Yaskawa INFORM job: A_ROOF_SIDE_0617_2_PAINT_36.JBI

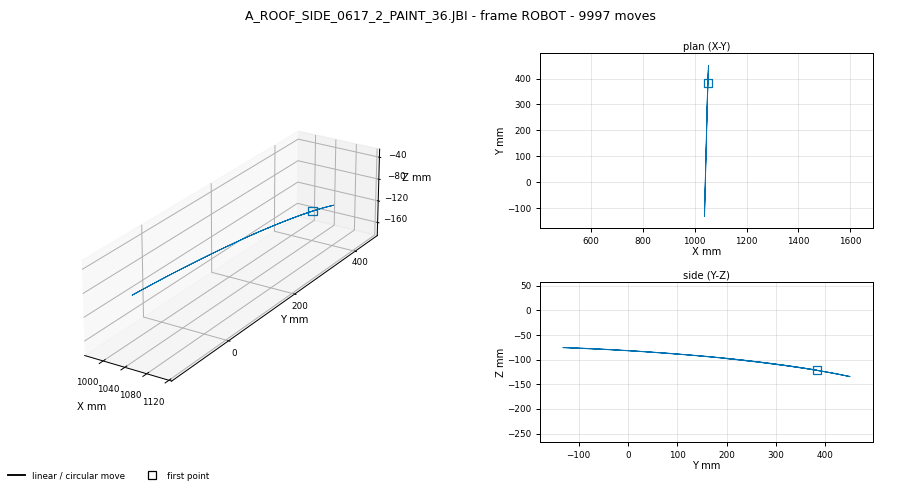
[picture p0: tool path of A_ROOF_SIDE_0617_2_PAINT_36.JBI in frame ROBOT, 9997 of 9997 moves have a stored position in this frame; points joined in program order, loops and branches not executed]
/JOB
//NAME A_ROOF_SIDE_0617_2_PAINT36
//POS
///NPOS 9997,0,0,0,0,0
///TOOL 1
///USER 0
///POSTYPE ROBOT
///RECTAN
///RCONF 1,0,0,0,0,0,0,0,0,0,0,0,0,0,0,0,0,0,0,0,0,0,0,0
C00000=1051.192,382.827,-120.850,173.969,40.523,157.828
C00001=1051.183,382.580,-120.809,173.963,40.517,157.826
C00002=1051.175,382.334,-120.768,173.957,40.511,157.824
C00003=1051.168,382.087,-120.727,173.951,40.505,157.822
C00004=1051.160,381.841,-120.686,173.945,40.499,157.821
C00005=1051.152,381.595,-120.645,173.938,40.493,157.819
C00006=1051.145,381.348,-120.604,173.932,40.487,157.817
C00007=1051.136,381.101,-120.563,173.926,40.481,157.815
C00008=1051.128,380.855,-120.523,173.919,40.475,157.814
C00009=1051.120,380.609,-120.482,173.913,40.469,157.812
C00010=1051.113,380.362,-120.441,173.908,40.463,157.810
C00011=1051.105,380.116,-120.400,173.901,40.458,157.809
C00012=1051.097,379.870,-120.359,173.895,40.452,157.807
C00013=1051.089,379.623,-120.319,173.889,40.446,157.805
C00014=1051.081,379.376,-120.279,173.882,40.440,157.804
C00015=1051.073,379.130,-120.238,173.877,40.434,157.802
C00016=1051.065,378.884,-120.198,173.871,40.429,157.800
C00017=1051.057,378.637,-120.158,173.864,40.423,157.798
C00018=1051.048,378.390,-120.117,173.858,40.417,157.797
C00019=1051.040,378.144,-120.076,173.853,40.412,157.795
C00020=1051.033,377.897,-120.036,173.847,40.406,157.794
C00021=1051.025,377.650,-119.995,173.840,40.400,157.792
C00022=1051.017,377.403,-119.956,173.834,40.395,157.790
C00023=1051.009,377.157,-119.915,173.829,40.389,157.789
C00024=1051.001,376.910,-119.875,173.823,40.383,157.787
C00025=1050.993,376.664,-119.834,173.817,40.378,157.785
C00026=1050.986,376.418,-119.795,173.810,40.372,157.784
C00027=1050.978,376.172,-119.754,173.805,40.367,157.782
C00028=1050.970,375.925,-119.714,173.799,40.361,157.780
C00029=1050.963,375.678,-119.674,173.793,40.356,157.779
C00030=1050.953,375.363,-119.623,173.785,40.348,157.777
C00031=1050.943,375.047,-119.571,173.778,40.341,157.775
C00032=1050.932,374.732,-119.520,173.771,40.334,157.773
C00033=1050.923,374.417,-119.469,173.763,40.327,157.771
C00034=1050.915,374.170,-119.429,173.757,40.321,157.769
C00035=1050.907,373.923,-119.389,173.751,40.316,157.768
C00036=1050.900,373.677,-119.349,173.746,40.310,157.766
C00037=1050.892,373.430,-119.309,173.740,40.305,157.764
C00038=1050.885,373.183,-119.269,173.734,40.300,157.763
C00039=1050.877,372.936,-119.229,173.729,40.294,157.761
C00040=1050.869,372.691,-119.190,173.723,40.288,157.760
C00041=1050.861,372.444,-119.150,173.717,40.283,157.758
C00042=1050.853,372.197,-119.110,173.711,40.278,157.757
C00043=1050.846,371.950,-119.070,173.705,40.272,157.755
C00044=1050.838,371.704,-119.031,173.699,40.267,157.753
C00045=1050.831,371.457,-118.991,173.694,40.262,157.752
C00046=1050.823,371.209,-118.951,173.688,40.256,157.750
C00047=1050.815,370.963,-118.912,173.683,40.251,157.749
C00048=1050.808,370.716,-118.873,173.677,40.246,157.747
C00049=1050.799,370.470,-118.833,173.672,40.240,157.746
C00050=1050.792,370.223,-118.793,173.666,40.235,157.744
C00051=1050.785,369.976,-118.754,173.660,40.230,157.743
C00052=1050.776,369.729,-118.715,173.655,40.225,157.741
C00053=1050.769,369.483,-118.675,173.649,40.219,157.740
C00054=1050.761,369.236,-118.637,173.644,40.214,157.738
C00055=1050.753,368.989,-118.597,173.638,40.209,157.737
C00056=1050.747,368.742,-118.558,173.633,40.204,157.735
C00057=1050.738,368.496,-118.519,173.627,40.199,157.734
C00058=1050.730,368.249,-118.479,173.621,40.193,157.732
C00059=1050.723,368.002,-118.441,173.616,40.188,157.731
C00060=1050.715,367.755,-118.401,173.610,40.183,157.729
C00061=1050.708,367.509,-118.362,173.605,40.178,157.728
C00062=1050.700,367.262,-118.323,173.599,40.173,157.727
C00063=1050.693,367.015,-118.284,173.594,40.167,157.725
C00064=1050.685,366.768,-118.245,173.588,40.163,157.724
C00065=1050.678,366.522,-118.206,173.583,40.157,157.722
C00066=1050.670,366.275,-118.167,173.577,40.152,157.721
C00067=1050.663,366.028,-118.128,173.572,40.147,157.719
C00068=1050.655,365.781,-118.088,173.566,40.142,157.718
C00069=1050.647,365.534,-118.050,173.561,40.137,157.716
C00070=1050.640,365.287,-118.011,173.555,40.132,157.715
C00071=1050.632,365.041,-117.972,173.551,40.127,157.714
C00072=1050.625,364.793,-117.933,173.545,40.122,157.712
C00073=1050.617,364.547,-117.894,173.540,40.117,157.711
C00074=1050.610,364.300,-117.856,173.534,40.111,157.709
C00075=1050.602,364.053,-117.817,173.529,40.107,157.708
C00076=1050.595,363.807,-117.777,173.523,40.101,157.706
C00077=1050.588,363.560,-117.739,173.518,40.097,157.705
C00078=1050.580,363.313,-117.700,173.512,40.091,157.704
C00079=1050.573,363.066,-117.662,173.508,40.086,157.702
C00080=1050.566,362.819,-117.623,173.503,40.082,157.701
C00081=1050.558,362.572,-117.584,173.497,40.077,157.699
C00082=1050.550,362.325,-117.546,173.492,40.071,157.698
C00083=1050.543,362.078,-117.507,173.486,40.067,157.697
C00084=1050.536,361.831,-117.469,173.481,40.062,157.695
C00085=1050.528,361.584,-117.431,173.477,40.057,157.694
C00086=1050.520,361.288,-117.385,173.470,40.051,157.692
C00087=1050.510,360.991,-117.338,173.463,40.045,157.691
C00088=1050.501,360.695,-117.293,173.458,40.039,157.689
C00089=1050.492,360.398,-117.246,173.451,40.034,157.687
C00090=1050.485,360.152,-117.208,173.445,40.029,157.686
C00091=1050.477,359.905,-117.170,173.441,40.024,157.685
C00092=1050.469,359.658,-117.132,173.436,40.019,157.683
C00093=1050.462,359.411,-117.094,173.430,40.014,157.682
C00094=1050.455,359.164,-117.055,173.425,40.010,157.681
C00095=1050.448,358.917,-117.017,173.421,40.005,157.679
C00096=1050.440,358.670,-116.979,173.415,40.000,157.678
C00097=1050.432,358.423,-116.941,173.410,39.995,157.677
C00098=1050.425,358.176,-116.903,173.404,39.990,157.675
C00099=1050.418,357.929,-116.865,173.400,39.986,157.674
C00100=1050.411,357.682,-116.827,173.395,39.981,157.673
C00101=1050.404,357.435,-116.789,173.389,39.976,157.671
C00102=1050.396,357.189,-116.751,173.384,39.972,157.670
C00103=1050.388,356.941,-116.713,173.380,39.967,157.669
C00104=1050.381,356.694,-116.675,173.374,39.963,157.667
C00105=1050.373,356.447,-116.637,173.369,39.958,157.666
C00106=1050.366,356.200,-116.600,173.365,39.953,157.665
C00107=1050.359,355.954,-116.561,173.360,39.949,157.664
C00108=1050.351,355.706,-116.524,173.354,39.944,157.662
C00109=1050.344,355.459,-116.486,173.349,39.939,157.661
C00110=1050.337,355.212,-116.449,173.345,39.935,157.660
C00111=1050.329,354.966,-116.411,173.339,39.930,157.658
C00112=1050.322,354.718,-116.373,173.334,39.925,157.657
C00113=1050.315,354.471,-116.336,173.330,39.921,157.656
C00114=1050.307,354.224,-116.298,173.324,39.916,157.655
C00115=1050.300,353.976,-116.260,173.319,39.912,157.653
C00116=1050.293,353.729,-116.223,173.315,39.907,157.652
C00117=1050.286,353.483,-116.185,173.310,39.903,157.651
C00118=1050.278,353.236,-116.147,173.305,39.898,157.650
C00119=1050.271,352.989,-116.110,173.300,39.893,157.648
C00120=1050.264,352.742,-116.072,173.295,39.889,157.647
C00121=1050.257,352.495,-116.035,173.290,39.884,157.646
C00122=1050.249,352.248,-115.997,173.285,39.879,157.644
C00123=1050.242,352.001,-115.960,173.281,39.875,157.643
C00124=1050.235,351.753,-115.922,173.276,39.871,157.642
C00125=1050.228,351.506,-115.885,173.270,39.866,157.641
C00126=1050.221,351.259,-115.848,173.266,39.862,157.640
C00127=1050.213,351.011,-115.810,173.261,39.857,157.638
C00128=1050.206,350.764,-115.773,173.257,39.853,157.637
C00129=1050.198,350.518,-115.736,173.251,39.848,157.636
C00130=1050.192,350.271,-115.699,173.246,39.844,157.635
C00131=1050.185,350.023,-115.662,173.242,39.839,157.633
C00132=1050.177,349.776,-115.624,173.237,39.835,157.632
C00133=1050.169,349.529,-115.587,173.232,39.830,157.631
C00134=1050.162,349.282,-115.550,173.227,39.826,157.630
C00135=1050.155,349.034,-115.513,173.223,39.822,157.629
C00136=1050.148,348.787,-115.475,173.218,39.818,157.627
C00137=1050.141,348.541,-115.439,173.214,39.813,157.626
C00138=1050.134,348.293,-115.402,173.208,39.808,157.625
C00139=1050.126,348.046,-115.365,173.204,39.804,157.624
C00140=1050.119,347.799,-115.328,173.199,39.800,157.623
C00141=1050.112,347.552,-115.291,173.194,39.796,157.621
C00142=1050.104,347.261,-115.247,173.188,39.791,157.620
C00143=1050.095,346.970,-115.204,173.183,39.785,157.619
C00144=1050.087,346.679,-115.160,173.178,39.780,157.617
C00145=1050.078,346.388,-115.117,173.172,39.775,157.616
C00146=1050.071,346.140,-115.081,173.168,39.771,157.615
C00147=1050.063,345.893,-115.044,173.163,39.767,157.614
C00148=1050.057,345.646,-115.007,173.159,39.763,157.612
C00149=1050.050,345.399,-114.970,173.154,39.758,157.611
C00150=1050.042,345.152,-114.933,173.149,39.754,157.610
C00151=1050.036,344.905,-114.897,173.144,39.750,157.609
C00152=1050.028,344.657,-114.861,173.140,39.745,157.608
C00153=1050.021,344.410,-114.823,173.135,39.741,157.606
C00154=1050.014,344.163,-114.787,173.131,39.737,157.605
C00155=1050.007,343.915,-114.751,173.126,39.733,157.604
C00156=1050.000,343.668,-114.714,173.122,39.729,157.603
C00157=1049.992,343.422,-114.677,173.117,39.724,157.602
C00158=1049.985,343.174,-114.640,173.112,39.720,157.601
C00159=1049.979,342.927,-114.604,173.108,39.716,157.600
C00160=1049.971,342.679,-114.568,173.103,39.712,157.599
C00161=1049.965,342.432,-114.531,173.099,39.707,157.597
C00162=1049.957,342.185,-114.495,173.095,39.703,157.596
C00163=1049.950,341.937,-114.459,173.090,39.699,157.595
C00164=1049.943,341.690,-114.422,173.085,39.695,157.594
C00165=1049.936,341.443,-114.386,173.080,39.691,157.593
C00166=1049.929,341.196,-114.350,173.076,39.687,157.592
C00167=1049.922,340.948,-114.314,173.072,39.683,157.591
C00168=1049.914,340.701,-114.277,173.067,39.679,157.590
C00169=1049.908,340.454,-114.241,173.063,39.674,157.588
C00170=1049.900,340.206,-114.205,173.058,39.671,157.587
C00171=1049.893,339.960,-114.169,173.054,39.666,157.586
C00172=1049.886,339.712,-114.132,173.050,39.662,157.585
C00173=1049.879,339.465,-114.096,173.045,39.658,157.584
C00174=1049.872,339.217,-114.061,173.040,39.654,157.583
C00175=1049.865,338.970,-114.024,173.036,39.650,157.582
C00176=1049.858,338.723,-113.988,173.031,39.646,157.581
C00177=1049.850,338.476,-113.952,173.027,39.642,157.580
C00178=1049.844,338.228,-113.916,173.023,39.638,157.579
C00179=1049.837,337.981,-113.880,173.018,39.634,157.577
C00180=1049.830,337.734,-113.844,173.014,39.630,157.576
C00181=1049.822,337.487,-113.808,173.010,39.626,157.575
C00182=1049.816,337.239,-113.772,173.005,39.622,157.574
C00183=1049.809,336.992,-113.737,173.001,39.617,157.573
C00184=1049.802,336.744,-113.701,172.997,39.614,157.572
C00185=1049.795,336.497,-113.665,172.993,39.610,157.571
C00186=1049.788,336.250,-113.628,172.988,39.605,157.570
C00187=1049.781,336.002,-113.593,172.984,39.602,157.569
C00188=1049.774,335.755,-113.557,172.980,39.598,157.568
C00189=1049.766,335.507,-113.522,172.975,39.594,157.567
C00190=1049.760,335.260,-113.485,172.970,39.590,157.566
C00191=1049.753,335.013,-113.450,172.966,39.586,157.565
C00192=1049.746,334.766,-113.414,172.962,39.582,157.564
C00193=1049.739,334.518,-113.379,172.957,39.578,157.562
C00194=1049.731,334.270,-113.343,172.953,39.574,157.561
C00195=1049.724,334.023,-113.308,172.949,39.570,157.560
C00196=1049.718,333.776,-113.272,172.945,39.566,157.559
C00197=1049.711,333.529,-113.237,172.940,39.563,157.558
C00198=1049.702,333.233,-113.195,172.935,39.558,157.557
C00199=1049.694,332.939,-113.152,172.931,39.553,157.556
C00200=1049.686,332.644,-113.109,172.926,39.549,157.555
C00201=1049.678,332.349,-113.068,172.920,39.544,157.553
C00202=1049.671,332.102,-113.032,172.916,39.540,157.552
C00203=1049.663,331.854,-112.996,172.911,39.536,157.551
C00204=1049.656,331.606,-112.961,172.907,39.533,157.550
C00205=1049.650,331.359,-112.926,172.903,39.529,157.549
C00206=1049.643,331.112,-112.891,172.899,39.525,157.548
C00207=1049.635,330.864,-112.855,172.895,39.521,157.547
C00208=1049.628,330.617,-112.820,172.890,39.517,157.546
C00209=1049.622,330.369,-112.785,172.887,39.513,157.545
C00210=1049.615,330.122,-112.749,172.883,39.510,157.544
C00211=1049.608,329.875,-112.714,172.879,39.506,157.543
C00212=1049.601,329.627,-112.679,172.875,39.502,157.542
C00213=1049.594,329.379,-112.644,172.871,39.498,157.541
C00214=1049.587,329.132,-112.609,172.866,39.494,157.540
C00215=1049.580,328.885,-112.574,172.862,39.491,157.539
C00216=1049.573,328.637,-112.539,172.858,39.487,157.538
C00217=1049.565,328.390,-112.504,172.854,39.483,157.537
C00218=1049.558,328.142,-112.469,172.850,39.480,157.536
C00219=1049.552,327.894,-112.434,172.846,39.476,157.535
C00220=1049.544,327.647,-112.400,172.841,39.472,157.534
C00221=1049.537,327.400,-112.365,172.837,39.469,157.533
C00222=1049.530,327.153,-112.330,172.833,39.465,157.532
C00223=1049.523,326.905,-112.296,172.829,39.461,157.531
C00224=1049.517,326.658,-112.261,172.825,39.457,157.530
C00225=1049.509,326.410,-112.226,172.821,39.454,157.529
C00226=1049.502,326.162,-112.191,172.817,39.450,157.528
C00227=1049.495,325.914,-112.156,172.812,39.446,157.527
C00228=1049.488,325.667,-112.122,172.808,39.443,157.526
C00229=1049.481,325.420,-112.086,172.804,39.439,157.525
C00230=1049.474,325.172,-112.053,172.800,39.435,157.524
C00231=1049.467,324.925,-112.017,172.797,39.432,157.524
C00232=1049.460,324.678,-111.982,172.793,39.428,157.523
C00233=1049.453,324.430,-111.949,172.789,39.424,157.522
C00234=1049.446,324.183,-111.913,172.785,39.421,157.521
C00235=1049.439,323.935,-111.880,172.781,39.417,157.520
C00236=1049.432,323.688,-111.844,172.777,39.414,157.519
C00237=1049.426,323.440,-111.809,172.772,39.410,157.518
C00238=1049.418,323.193,-111.775,172.768,39.406,157.517
C00239=1049.412,322.945,-111.740,172.764,39.403,157.516
C00240=1049.404,322.697,-111.707,172.760,39.399,157.515
C00241=1049.398,322.450,-111.671,172.756,39.396,157.514
C00242=1049.391,322.202,-111.637,172.752,39.392,157.513
C00243=1049.384,321.954,-111.603,172.748,39.388,157.512
C00244=1049.377,321.707,-111.568,172.745,39.385,157.511
C00245=1049.370,321.459,-111.534,172.741,39.381,157.510
C00246=1049.364,321.213,-111.499,172.737,39.378,157.509
C00247=1049.357,320.965,-111.466,172.733,39.374,157.508
C00248=1049.350,320.717,-111.431,172.729,39.371,157.507
C00249=1049.343,320.470,-111.397,172.725,39.367,157.506
C00250=1049.336,320.222,-111.362,172.721,39.363,157.506
C00251=1049.330,319.974,-111.328,172.717,39.360,157.504
C00252=1049.322,319.727,-111.293,172.713,39.356,157.504
C00253=1049.316,319.480,-111.259,172.709,39.352,157.503
C00254=1049.308,319.180,-111.218,172.704,39.349,157.502
C00255=1049.299,318.880,-111.176,172.700,39.344,157.500
C00256=1049.292,318.580,-111.135,172.695,39.340,157.499
C00257=1049.283,318.280,-111.093,172.691,39.335,157.498
C00258=1049.277,318.032,-111.059,172.687,39.332,157.497
C00259=1049.269,317.784,-111.025,172.683,39.328,157.496
C00260=1049.264,317.537,-110.991,172.680,39.325,157.495
C00261=1049.256,317.289,-110.957,172.676,39.321,157.494
C00262=1049.250,317.041,-110.923,172.672,39.318,157.494
C00263=1049.242,316.794,-110.888,172.668,39.314,157.493
C00264=1049.236,316.547,-110.854,172.664,39.311,157.492
C00265=1049.229,316.299,-110.820,172.660,39.307,157.491
C00266=1049.223,316.051,-110.786,172.656,39.303,157.490
C00267=1049.216,315.804,-110.752,172.652,39.300,157.489
C00268=1049.210,315.556,-110.718,172.649,39.297,157.488
C00269=1049.203,315.308,-110.684,172.645,39.293,157.487
C00270=1049.197,315.061,-110.650,172.641,39.290,157.486
C00271=1049.189,314.813,-110.616,172.637,39.286,157.485
C00272=1049.184,314.566,-110.582,172.634,39.282,157.484
C00273=1049.176,314.319,-110.548,172.630,39.279,157.484
C00274=1049.170,314.071,-110.514,172.626,39.276,157.483
C00275=1049.163,313.824,-110.480,172.622,39.272,157.482
C00276=1049.157,313.576,-110.446,172.619,39.269,157.481
C00277=1049.151,313.328,-110.413,172.615,39.265,157.480
C00278=1049.144,313.080,-110.379,172.611,39.261,157.479
C00279=1049.137,312.832,-110.345,172.607,39.258,157.478
C00280=1049.130,312.585,-110.312,172.603,39.255,157.477
C00281=1049.123,312.337,-110.278,172.600,39.251,157.476
C00282=1049.116,312.089,-110.245,172.597,39.248,157.476
C00283=1049.110,311.842,-110.211,172.593,39.245,157.475
C00284=1049.103,311.594,-110.178,172.589,39.241,157.474
C00285=1049.096,311.346,-110.144,172.585,39.238,157.473
C00286=1049.089,311.099,-110.111,172.581,39.235,157.472
C00287=1049.081,310.852,-110.078,172.578,39.232,157.471
C00288=1049.074,310.604,-110.044,172.574,39.228,157.470
C00289=1049.068,310.356,-110.012,172.570,39.225,157.470
C00290=1049.061,310.109,-109.978,172.566,39.222,157.469
C00291=1049.054,309.862,-109.944,172.563,39.218,157.468
C00292=1049.047,309.613,-109.911,172.560,39.215,157.467
C00293=1049.041,309.366,-109.878,172.556,39.212,157.466
C00294=1049.034,309.118,-109.845,172.552,39.208,157.465
C00295=1049.026,308.870,-109.811,172.548,39.205,157.464
C00296=1049.020,308.623,-109.778,172.544,39.202,157.464
C00297=1049.013,308.374,-109.745,172.541,39.198,157.463
C00298=1049.006,308.128,-109.712,172.538,39.195,157.462
C00299=1048.999,307.880,-109.679,172.534,39.192,157.461
C00300=1048.992,307.633,-109.646,172.530,39.188,157.460
C00301=1048.986,307.384,-109.613,172.526,39.185,157.459
C00302=1048.979,307.137,-109.579,172.523,39.182,157.458
C00303=1048.972,306.889,-109.546,172.519,39.179,157.458
C00304=1048.966,306.641,-109.513,172.516,39.176,157.457
C00305=1048.959,306.394,-109.480,172.512,39.172,157.456
C00306=1048.952,306.146,-109.447,172.508,39.169,157.455
C00307=1048.945,305.899,-109.415,172.505,39.166,157.454
C00308=1048.938,305.651,-109.381,172.501,39.162,157.453
C00309=1048.932,305.404,-109.348,172.498,39.159,157.453
C00310=1048.924,305.108,-109.308,172.493,39.155,157.452
C00311=1048.916,304.812,-109.269,172.489,39.151,157.451
C00312=1048.908,304.516,-109.230,172.485,39.147,157.450
C00313=1048.899,304.221,-109.191,172.480,39.143,157.449
C00314=1048.893,303.973,-109.158,172.478,39.140,157.448
C00315=1048.886,303.726,-109.125,172.474,39.137,157.447
C00316=1048.880,303.478,-109.092,172.470,39.134,157.446
C00317=1048.873,303.230,-109.059,172.466,39.131,157.445
C00318=1048.867,302.983,-109.026,172.463,39.127,157.444
C00319=1048.860,302.734,-108.993,172.460,39.124,157.444
C00320=1048.853,302.487,-108.961,172.456,39.121,157.443
C00321=1048.847,302.239,-108.928,172.452,39.117,157.442
C00322=1048.840,301.991,-108.895,172.449,39.114,157.441
C00323=1048.834,301.743,-108.862,172.446,39.111,157.440
C00324=1048.827,301.496,-108.830,172.442,39.108,157.439
C00325=1048.820,301.249,-108.797,172.439,39.104,157.439
C00326=1048.813,301.000,-108.764,172.435,39.101,157.438
C00327=1048.807,300.753,-108.732,172.431,39.098,157.437
C00328=1048.801,300.505,-108.699,172.428,39.095,157.436
C00329=1048.794,300.258,-108.666,172.425,39.092,157.435
C00330=1048.788,300.009,-108.633,172.421,39.088,157.435
C00331=1048.781,299.762,-108.601,172.417,39.085,157.434
C00332=1048.774,299.514,-108.568,172.415,39.082,157.433
C00333=1048.768,299.267,-108.535,172.411,39.079,157.432
C00334=1048.762,299.019,-108.503,172.407,39.075,157.431
C00335=1048.755,298.771,-108.469,172.404,39.072,157.430
C00336=1048.748,298.524,-108.437,172.401,39.069,157.430
C00337=1048.742,298.275,-108.405,172.397,39.066,157.429
C00338=1048.735,298.028,-108.373,172.394,39.062,157.428
C00339=1048.729,297.780,-108.340,172.390,39.059,157.427
C00340=1048.723,297.533,-108.307,172.387,39.056,157.426
C00341=1048.715,297.285,-108.275,172.384,39.053,157.426
C00342=1048.709,297.036,-108.243,172.380,39.050,157.425
C00343=1048.703,296.789,-108.210,172.377,39.046,157.424
C00344=1048.697,296.541,-108.177,172.374,39.043,157.423
C00345=1048.690,296.294,-108.145,172.370,39.040,157.422
C00346=1048.684,296.046,-108.113,172.367,39.037,157.422
C00347=1048.677,295.798,-108.080,172.363,39.033,157.421
C00348=1048.670,295.550,-108.048,172.360,39.031,157.420
C00349=1048.664,295.302,-108.016,172.357,39.027,157.419
C00350=1048.657,295.055,-107.983,172.353,39.024,157.418
C00351=1048.651,294.806,-107.951,172.351,39.021,157.418
C00352=1048.644,294.559,-107.919,172.347,39.018,157.417
C00353=1048.638,294.311,-107.887,172.343,39.015,157.416
C00354=1048.631,294.064,-107.855,172.340,39.011,157.415
C00355=1048.623,293.815,-107.823,172.337,39.009,157.415
C00356=1048.617,293.567,-107.791,172.333,39.005,157.414
C00357=1048.610,293.320,-107.759,172.330,39.003,157.413
C00358=1048.604,293.072,-107.726,172.326,38.999,157.412
C00359=1048.597,292.824,-107.695,172.324,38.996,157.411
C00360=1048.590,292.577,-107.663,172.320,38.993,157.411
C00361=1048.584,292.329,-107.631,172.316,38.990,157.410
C00362=1048.578,292.081,-107.599,172.314,38.987,157.409
C00363=1048.571,291.833,-107.567,172.310,38.984,157.408
C00364=1048.565,291.585,-107.535,172.307,38.981,157.407
C00365=1048.558,291.337,-107.504,172.304,38.978,157.407
C00366=1048.550,291.058,-107.467,172.300,38.975,157.406
C00367=1048.542,290.778,-107.431,172.296,38.971,157.405
C00368=1048.535,290.499,-107.396,172.292,38.967,157.404
C00369=1048.527,290.219,-107.360,172.289,38.964,157.403
C00370=1048.521,289.971,-107.328,172.286,38.961,157.403
C00371=1048.514,289.723,-107.296,172.282,38.958,157.402
C00372=1048.507,289.476,-107.264,172.279,38.955,157.401
C00373=1048.501,289.228,-107.232,172.276,38.951,157.400
C00374=1048.495,288.980,-107.201,172.273,38.949,157.399
C00375=1048.488,288.732,-107.169,172.269,38.946,157.399
C00376=1048.481,288.484,-107.138,172.266,38.942,157.398
C00377=1048.475,288.236,-107.106,172.263,38.940,157.397
C00378=1048.468,287.988,-107.073,172.260,38.936,157.396
C00379=1048.461,287.741,-107.042,172.256,38.933,157.396
C00380=1048.455,287.493,-107.011,172.254,38.931,157.395
C00381=1048.449,287.245,-106.980,172.250,38.927,157.394
C00382=1048.442,286.998,-106.948,172.247,38.924,157.393
C00383=1048.435,286.750,-106.917,172.244,38.922,157.393
C00384=1048.429,286.501,-106.885,172.240,38.918,157.392
C00385=1048.422,286.254,-106.853,172.237,38.915,157.391
C00386=1048.416,286.006,-106.822,172.234,38.913,157.391
C00387=1048.409,285.758,-106.790,172.231,38.909,157.390
C00388=1048.402,285.510,-106.759,172.227,38.906,157.389
C00389=1048.396,285.262,-106.728,172.225,38.904,157.388
C00390=1048.389,285.014,-106.696,172.221,38.900,157.387
C00391=1048.382,284.766,-106.665,172.218,38.897,157.387
C00392=1048.376,284.518,-106.634,172.215,38.895,157.386
C00393=1048.369,284.270,-106.602,172.212,38.891,157.385
C00394=1048.362,284.022,-106.571,172.208,38.888,157.385
C00395=1048.356,283.774,-106.540,172.206,38.886,157.384
C00396=1048.349,283.527,-106.509,172.203,38.883,157.383
C00397=1048.343,283.279,-106.477,172.199,38.879,157.382
C00398=1048.336,283.031,-106.446,172.197,38.877,157.382
C00399=1048.330,282.782,-106.415,172.193,38.874,157.381
C00400=1048.323,282.534,-106.384,172.190,38.870,157.380
C00401=1048.316,282.287,-106.352,172.187,38.868,157.379
C00402=1048.309,282.039,-106.321,172.184,38.865,157.379
C00403=1048.304,281.791,-106.290,172.180,38.862,157.378
C00404=1048.297,281.543,-106.259,172.178,38.858,157.377
C00405=1048.290,281.295,-106.227,172.175,38.856,157.376
C00406=1048.283,281.047,-106.196,172.171,38.853,157.376
C00407=1048.277,280.799,-106.165,172.169,38.849,157.375
C00408=1048.271,280.551,-106.134,172.165,38.847,157.374
C00409=1048.264,280.303,-106.103,172.162,38.844,157.374
C00410=1048.258,280.055,-106.072,172.159,38.841,157.373
C00411=1048.251,279.807,-106.041,172.156,38.838,157.372
C00412=1048.244,279.559,-106.009,172.153,38.835,157.371
C00413=1048.238,279.311,-105.979,172.150,38.832,157.371
C00414=1048.232,279.063,-105.947,172.147,38.829,157.370
C00415=1048.225,278.815,-105.917,172.143,38.826,157.369
C00416=1048.219,278.567,-105.885,172.141,38.823,157.368
C00417=1048.212,278.319,-105.856,172.138,38.820,157.368
C00418=1048.205,278.072,-105.824,172.134,38.817,157.367
C00419=1048.199,277.823,-105.793,172.132,38.814,157.366
C00420=1048.192,277.575,-105.762,172.128,38.812,157.366
C00421=1048.186,277.327,-105.732,172.126,38.809,157.365
C00422=1048.179,277.059,-105.698,172.122,38.805,157.364
C00423=1048.171,276.791,-105.665,172.119,38.802,157.363
C00424=1048.164,276.524,-105.632,172.115,38.799,157.363
C00425=1048.157,276.255,-105.599,172.113,38.796,157.362
C00426=1048.151,276.007,-105.568,172.109,38.793,157.361
C00427=1048.144,275.759,-105.537,172.106,38.790,157.360
C00428=1048.138,275.512,-105.506,172.104,38.787,157.360
C00429=1048.131,275.263,-105.476,172.100,38.784,157.359
C00430=1048.125,275.015,-105.445,172.097,38.781,157.358
C00431=1048.118,274.768,-105.414,172.095,38.778,157.357
C00432=1048.111,274.519,-105.384,172.091,38.775,157.357
C00433=1048.105,274.271,-105.353,172.089,38.772,157.356
C00434=1048.099,274.023,-105.323,172.086,38.769,157.355
C00435=1048.092,273.776,-105.292,172.082,38.767,157.355
C00436=1048.085,273.527,-105.261,172.080,38.764,157.354
C00437=1048.079,273.279,-105.231,172.077,38.761,157.353
C00438=1048.072,273.031,-105.201,172.073,38.758,157.353
C00439=1048.066,272.782,-105.170,172.071,38.755,157.352
C00440=1048.060,272.535,-105.139,172.068,38.752,157.351
C00441=1048.052,272.287,-105.109,172.065,38.749,157.350
C00442=1048.047,272.039,-105.078,172.062,38.746,157.350
C00443=1048.040,271.791,-105.048,172.059,38.743,157.349
C00444=1048.033,271.542,-105.018,172.056,38.740,157.348
C00445=1048.027,271.295,-104.987,172.053,38.738,157.348
C00446=1048.020,271.046,-104.957,172.050,38.735,157.347
C00447=1048.014,270.798,-104.926,172.047,38.732,157.346
C00448=1048.007,270.551,-104.896,172.044,38.729,157.346
C00449=1048.000,270.302,-104.865,172.042,38.726,157.345
C00450=1047.994,270.055,-104.835,172.038,38.723,157.344
C00451=1047.987,269.806,-104.805,172.035,38.721,157.343
C00452=1047.980,269.558,-104.775,172.033,38.718,157.343
C00453=1047.974,269.310,-104.744,172.030,38.715,157.342
C00454=1047.967,269.062,-104.714,172.027,38.712,157.341
C00455=1047.961,268.814,-104.684,172.024,38.709,157.341
C00456=1047.955,268.566,-104.654,172.021,38.706,157.340
C00457=1047.949,268.318,-104.624,172.019,38.703,157.339
C00458=1047.942,268.070,-104.594,172.015,38.700,157.338
C00459=1047.936,267.822,-104.564,172.012,38.697,157.338
C00460=1047.929,267.573,-104.533,172.010,38.694,157.337
C00461=1047.922,267.325,-104.503,172.007,38.691,157.336
C00462=1047.916,267.077,-104.473,172.004,38.689,157.336
C00463=1047.909,266.829,-104.443,172.001,38.686,157.335
C00464=1047.903,266.581,-104.413,171.998,38.683,157.334
C00465=1047.896,266.333,-104.383,171.995,38.680,157.334
C00466=1047.889,266.085,-104.353,171.992,38.678,157.333
C00467=1047.883,265.837,-104.323,171.990,38.675,157.332
C00468=1047.876,265.589,-104.293,171.987,38.672,157.332
C00469=1047.869,265.340,-104.263,171.984,38.669,157.331
C00470=1047.864,265.092,-104.233,171.981,38.666,157.330
C00471=1047.857,264.844,-104.203,171.978,38.663,157.330
C00472=1047.850,264.597,-104.173,171.976,38.661,157.329
C00473=1047.844,264.347,-104.143,171.973,38.658,157.328
C00474=1047.837,264.100,-104.113,171.969,38.655,157.328
C00475=1047.831,263.852,-104.084,171.967,38.652,157.327
C00476=1047.825,263.603,-104.054,171.964,38.649,157.326
C00477=1047.818,263.356,-104.024,171.962,38.646,157.326
C00478=1047.811,263.092,-103.992,171.959,38.643,157.325
C00479=1047.804,262.829,-103.960,171.955,38.640,157.324
C00480=1047.798,262.565,-103.929,171.953,38.637,157.323
C00481=1047.790,262.301,-103.897,171.950,38.634,157.323
C00482=1047.784,262.053,-103.868,171.946,38.631,157.322
C00483=1047.777,261.804,-103.838,171.944,38.628,157.321
C00484=1047.770,261.557,-103.808,171.941,38.626,157.321
C00485=1047.764,261.308,-103.779,171.939,38.623,157.320
C00486=1047.757,261.061,-103.749,171.935,38.620,157.319
C00487=1047.750,260.812,-103.720,171.933,38.618,157.319
C00488=1047.744,260.564,-103.690,171.930,38.615,157.318
C00489=1047.737,260.315,-103.661,171.927,38.612,157.317
C00490=1047.730,260.068,-103.631,171.925,38.609,157.317
C00491=1047.723,259.820,-103.603,171.921,38.606,157.316
C00492=1047.716,259.571,-103.573,171.919,38.604,157.315
C00493=1047.710,259.324,-103.543,171.916,38.601,157.315
C00494=1047.703,259.075,-103.514,171.913,38.598,157.314
C00495=1047.697,258.827,-103.485,171.911,38.595,157.313
C00496=1047.690,258.578,-103.455,171.908,38.592,157.313
C00497=1047.683,258.330,-103.426,171.905,38.589,157.312
C00498=1047.677,258.082,-103.397,171.902,38.587,157.311
C00499=1047.670,257.834,-103.367,171.900,38.584,157.311
C00500=1047.664,257.586,-103.338,171.897,38.581,157.310
C00501=1047.657,257.338,-103.309,171.894,38.579,157.309
C00502=1047.650,257.090,-103.278,171.892,38.576,157.309
C00503=1047.644,256.841,-103.249,171.889,38.573,157.308
C00504=1047.638,256.593,-103.220,171.886,38.571,157.308
C00505=1047.631,256.344,-103.191,171.883,38.568,157.307
C00506=1047.624,256.097,-103.161,171.881,38.565,157.306
C00507=1047.618,255.849,-103.132,171.878,38.562,157.305
C00508=1047.611,255.600,-103.103,171.875,38.559,157.305
C00509=1047.605,255.352,-103.074,171.873,38.556,157.304
C00510=1047.598,255.104,-103.045,171.870,38.553,157.303
C00511=1047.591,254.856,-103.015,171.868,38.551,157.303
C00512=1047.585,254.608,-102.986,171.865,38.548,157.302
C00513=1047.578,254.360,-102.957,171.861,38.545,157.302
C00514=1047.572,254.111,-102.928,171.859,38.542,157.301
C00515=1047.565,253.863,-102.899,171.856,38.539,157.300
C00516=1047.559,253.614,-102.870,171.854,38.536,157.299
C00517=1047.553,253.366,-102.840,171.851,38.534,157.299
C00518=1047.546,253.117,-102.811,171.849,38.531,157.298
C00519=1047.539,252.870,-102.781,171.846,38.528,157.298
C00520=1047.533,252.622,-102.752,171.843,38.526,157.297
C00521=1047.526,252.374,-102.724,171.841,38.523,157.296
C00522=1047.520,252.126,-102.695,171.838,38.520,157.296
C00523=1047.513,251.877,-102.665,171.836,38.517,157.295
C00524=1047.507,251.629,-102.636,171.833,38.514,157.294
C00525=1047.501,251.381,-102.607,171.831,38.511,157.294
C00526=1047.494,251.133,-102.578,171.828,38.509,157.293
C00527=1047.488,250.885,-102.549,171.825,38.506,157.292
C00528=1047.481,250.636,-102.520,171.822,38.503,157.292
C00529=1047.475,250.388,-102.491,171.819,38.500,157.291
C00530=1047.469,250.139,-102.462,171.817,38.497,157.290
C00531=1047.462,249.892,-102.433,171.814,38.494,157.290
C00532=1047.456,249.643,-102.405,171.812,38.491,157.289
C00533=1047.449,249.395,-102.376,171.809,38.489,157.288
C00534=1047.442,249.129,-102.345,171.806,38.486,157.288
C00535=1047.435,248.864,-102.314,171.804,38.483,157.287
C00536=1047.428,248.599,-102.283,171.801,38.480,157.286
C00537=1047.422,248.334,-102.252,171.799,38.476,157.285
C00538=1047.416,248.086,-102.223,171.796,38.474,157.285
C00539=1047.409,247.837,-102.194,171.793,38.471,157.284
C00540=1047.403,247.589,-102.165,171.791,38.468,157.284
C00541=1047.397,247.341,-102.136,171.788,38.465,157.283
C00542=1047.391,247.093,-102.107,171.786,38.462,157.282
C00543=1047.384,246.844,-102.078,171.783,38.459,157.281
C00544=1047.377,246.596,-102.050,171.781,38.457,157.281
C00545=1047.371,246.348,-102.021,171.778,38.454,157.280
C00546=1047.365,246.099,-101.992,171.775,38.451,157.279
C00547=1047.358,245.851,-101.963,171.773,38.448,157.279
C00548=1047.352,245.603,-101.935,171.770,38.445,157.278
C00549=1047.345,245.355,-101.906,171.768,38.443,157.278
C00550=1047.339,245.107,-101.877,171.765,38.440,157.277
C00551=1047.333,244.858,-101.849,171.763,38.437,157.276
C00552=1047.326,244.610,-101.820,171.760,38.434,157.276
C00553=1047.320,244.362,-101.791,171.757,38.431,157.275
C00554=1047.313,244.113,-101.764,171.755,38.428,157.274
C00555=1047.307,243.865,-101.735,171.752,38.426,157.274
C00556=1047.301,243.617,-101.706,171.750,38.423,157.273
C00557=1047.294,243.368,-101.678,171.747,38.420,157.272
C00558=1047.287,243.120,-101.648,171.745,38.417,157.272
C00559=1047.281,242.872,-101.621,171.742,38.414,157.271
C00560=1047.274,242.623,-101.592,171.741,38.412,157.270
C00561=1047.268,242.375,-101.563,171.738,38.409,157.270
C00562=1047.261,242.127,-101.535,171.735,38.406,157.269
C00563=1047.255,241.878,-101.507,171.733,38.403,157.268
C00564=1047.248,241.630,-101.478,171.730,38.400,157.268
C00565=1047.243,241.381,-101.450,171.728,38.397,157.267
C00566=1047.236,241.134,-101.421,171.725,38.395,157.267
C00567=1047.230,240.885,-101.393,171.723,38.392,157.266
C00568=1047.223,240.637,-101.365,171.720,38.389,157.265
C00569=1047.216,240.389,-101.337,171.718,38.386,157.265
C00570=1047.210,240.140,-101.309,171.715,38.384,157.264
C00571=1047.203,239.892,-101.280,171.713,38.381,157.263
C00572=1047.197,239.643,-101.252,171.710,38.378,157.263
C00573=1047.190,239.395,-101.224,171.707,38.375,157.262
C00574=1047.183,239.147,-101.196,171.706,38.373,157.261
C00575=1047.177,238.898,-101.167,171.703,38.370,157.261
C00576=1047.171,238.650,-101.140,171.701,38.367,157.260
C00577=1047.164,238.402,-101.111,171.698,38.364,157.259
C00578=1047.158,238.153,-101.083,171.696,38.361,157.259
C00579=1047.151,237.905,-101.055,171.693,38.359,157.258
C00580=1047.144,237.657,-101.027,171.691,38.356,157.258
C00581=1047.138,237.408,-100.998,171.688,38.353,157.257
C00582=1047.132,237.160,-100.971,171.686,38.350,157.256
C00583=1047.125,236.911,-100.943,171.683,38.348,157.256
C00584=1047.118,236.664,-100.914,171.682,38.345,157.255
C00585=1047.112,236.415,-100.886,171.679,38.342,157.254
C00586=1047.105,236.166,-100.858,171.676,38.339,157.254
C00587=1047.099,235.918,-100.831,171.674,38.337,157.253
C00588=1047.093,235.670,-100.803,171.671,38.334,157.252
C00589=1047.086,235.422,-100.774,171.669,38.331,157.252
C00590=1047.078,235.151,-100.744,171.666,38.328,157.251
C00591=1047.072,234.879,-100.714,171.664,38.325,157.250
C00592=1047.065,234.609,-100.684,171.661,38.322,157.250
C00593=1047.058,234.337,-100.652,171.658,38.319,157.249
C00594=1047.052,234.089,-100.625,171.656,38.316,157.248
C00595=1047.045,233.841,-100.597,171.653,38.313,157.248
C00596=1047.039,233.593,-100.568,171.652,38.310,157.247
C00597=1047.032,233.344,-100.541,171.649,38.307,157.246
C00598=1047.025,233.096,-100.513,171.647,38.305,157.246
C00599=1047.019,232.847,-100.485,171.644,38.302,157.245
C00600=1047.013,232.599,-100.457,171.642,38.299,157.244
C00601=1047.007,232.351,-100.429,171.639,38.296,157.244
C00602=1047.000,232.102,-100.402,171.638,38.293,157.243
C00603=1046.993,231.854,-100.374,171.635,38.290,157.243
C00604=1046.987,231.606,-100.346,171.632,38.288,157.242
C00605=1046.980,231.357,-100.319,171.630,38.285,157.241
C00606=1046.973,231.109,-100.291,171.627,38.282,157.241
C00607=1046.967,230.860,-100.262,171.626,38.279,157.240
C00608=1046.961,230.612,-100.235,171.623,38.276,157.239
C00609=1046.955,230.364,-100.207,171.621,38.273,157.239
C00610=1046.948,230.115,-100.180,171.618,38.271,157.238
C00611=1046.941,229.867,-100.152,171.616,38.268,157.238
C00612=1046.935,229.618,-100.125,171.614,38.265,157.237
C00613=1046.929,229.370,-100.098,171.612,38.262,157.236
C00614=1046.922,229.122,-100.070,171.609,38.259,157.236
C00615=1046.915,228.873,-100.042,171.607,38.257,157.235
C00616=1046.909,228.625,-100.014,171.604,38.254,157.234
C00617=1046.902,228.376,-99.987,171.603,38.251,157.234
C00618=1046.896,228.128,-99.960,171.600,38.248,157.233
C00619=1046.890,227.879,-99.932,171.598,38.246,157.232
C00620=1046.883,227.631,-99.904,171.595,38.243,157.232
C00621=1046.876,227.383,-99.877,171.593,38.240,157.231
C00622=1046.870,227.134,-99.850,171.591,38.237,157.230
C00623=1046.863,226.885,-99.822,171.588,38.235,157.230
C00624=1046.857,226.637,-99.795,171.586,38.232,157.229
C00625=1046.850,226.389,-99.768,171.583,38.229,157.229
C00626=1046.843,226.140,-99.741,171.582,38.226,157.228
C00627=1046.837,225.892,-99.713,171.579,38.224,157.227
C00628=1046.831,225.644,-99.685,171.577,38.221,157.227
C00629=1046.824,225.395,-99.658,171.574,38.218,157.226
C00630=1046.817,225.146,-99.631,171.573,38.215,157.225
C00631=1046.811,224.898,-99.603,171.570,38.212,157.225
C00632=1046.805,224.650,-99.576,171.568,38.209,157.224
C00633=1046.798,224.401,-99.549,171.565,38.207,157.224
C00634=1046.791,224.153,-99.521,171.564,38.204,157.223
C00635=1046.785,223.904,-99.494,171.561,38.201,157.222
C00636=1046.778,223.656,-99.467,171.559,38.198,157.222
C00637=1046.772,223.407,-99.440,171.557,38.195,157.221
C00638=1046.765,223.159,-99.412,171.554,38.192,157.220
C00639=1046.759,222.911,-99.385,171.552,38.189,157.220
C00640=1046.753,222.662,-99.358,171.549,38.187,157.219
C00641=1046.746,222.414,-99.331,171.548,38.184,157.219
C00642=1046.740,222.166,-99.304,171.545,38.181,157.218
C00643=1046.733,221.917,-99.276,171.543,38.178,157.217
C00644=1046.727,221.668,-99.249,171.541,38.175,157.217
C00645=1046.721,221.420,-99.222,171.539,38.173,157.216
C00646=1046.714,221.141,-99.191,171.536,38.169,157.215
C00647=1046.706,220.863,-99.162,171.534,38.166,157.215
C00648=1046.699,220.585,-99.131,171.531,38.163,157.214
C00649=1046.692,220.306,-99.100,171.528,38.160,157.213
C00650=1046.685,220.057,-99.074,171.527,38.157,157.212
C00651=1046.679,219.810,-99.046,171.524,38.154,157.212
C00652=1046.671,219.561,-99.020,171.522,38.152,157.211
C00653=1046.665,219.312,-98.993,171.520,38.149,157.211
C00654=1046.659,219.064,-98.966,171.518,38.146,157.210
C00655=1046.652,218.815,-98.939,171.515,38.143,157.209
C00656=1046.646,218.566,-98.912,171.514,38.140,157.209
C00657=1046.639,218.319,-98.885,171.511,38.138,157.208
C00658=1046.632,218.070,-98.858,171.509,38.135,157.207
C00659=1046.626,217.821,-98.831,171.507,38.132,157.207
C00660=1046.619,217.573,-98.805,171.505,38.129,157.206
C00661=1046.613,217.324,-98.777,171.502,38.126,157.206
C00662=1046.606,217.075,-98.751,171.501,38.123,157.205
C00663=1046.600,216.827,-98.724,171.498,38.120,157.204
C00664=1046.592,216.579,-98.697,171.496,38.118,157.204
C00665=1046.587,216.331,-98.671,171.494,38.115,157.203
C00666=1046.580,216.082,-98.644,171.492,38.112,157.202
C00667=1046.574,215.834,-98.618,171.489,38.109,157.202
C00668=1046.567,215.585,-98.590,171.488,38.106,157.201
C00669=1046.560,215.336,-98.563,171.485,38.104,157.201
C00670=1046.554,215.088,-98.537,171.483,38.101,157.200
C00671=1046.547,214.839,-98.510,171.481,38.098,157.199
C00672=1046.541,214.591,-98.483,171.479,38.095,157.199
C00673=1046.535,214.342,-98.456,171.477,38.092,157.198
C00674=1046.528,214.094,-98.430,171.474,38.089,157.197
C00675=1046.522,213.845,-98.403,171.472,38.087,157.197
C00676=1046.515,213.597,-98.377,171.471,38.084,157.196
C00677=1046.509,213.348,-98.350,171.468,38.081,157.196
C00678=1046.502,213.100,-98.324,171.466,38.078,157.195
C00679=1046.496,212.852,-98.296,171.464,38.075,157.194
C00680=1046.489,212.604,-98.270,171.461,38.072,157.194
C00681=1046.483,212.355,-98.243,171.460,38.069,157.193
C00682=1046.477,212.106,-98.216,171.457,38.067,157.192
C00683=1046.470,211.857,-98.190,171.456,38.064,157.192
C00684=1046.463,211.609,-98.164,171.453,38.061,157.191
C00685=1046.457,211.360,-98.137,171.451,38.058,157.190
C00686=1046.450,211.112,-98.110,171.449,38.055,157.190
C00687=1046.444,210.863,-98.084,171.447,38.052,157.189
C00688=1046.437,210.615,-98.057,171.445,38.049,157.189
C00689=1046.431,210.366,-98.031,171.443,38.046,157.188
C00690=1046.424,210.117,-98.004,171.441,38.043,157.187
C00691=1046.418,209.869,-97.978,171.439,38.040,157.187
C00692=1046.412,209.621,-97.952,171.436,38.037,157.186
C00693=1046.405,209.372,-97.925,171.435,38.035,157.185
C00694=1046.398,209.124,-97.899,171.432,38.032,157.185
C00695=1046.391,208.875,-97.873,171.431,38.029,157.184
C00696=1046.385,208.627,-97.846,171.428,38.026,157.183
C00697=1046.378,208.378,-97.820,171.427,38.023,157.183
C00698=1046.372,208.130,-97.794,171.424,38.021,157.182
C00699=1046.366,207.881,-97.767,171.422,38.018,157.182
C00700=1046.359,207.633,-97.741,171.420,38.015,157.181
C00701=1046.352,207.384,-97.715,171.418,38.012,157.180
C00702=1046.345,207.111,-97.686,171.416,38.009,157.180
C00703=1046.338,206.838,-97.657,171.414,38.005,157.179
C00704=1046.331,206.565,-97.628,171.411,38.002,157.178
C00705=1046.324,206.292,-97.600,171.409,37.999,157.178
C00706=1046.297,205.240,-97.493,171.157,37.900,157.153
C00707=1046.291,204.992,-97.468,171.155,37.897,157.152
C00708=1046.285,204.743,-97.443,171.151,37.896,157.152
C00709=1046.279,204.495,-97.418,171.149,37.893,157.152
C00710=1046.273,204.245,-97.393,171.147,37.891,157.151
C00711=1046.267,203.997,-97.368,171.143,37.889,157.151
C00712=1046.261,203.748,-97.342,171.141,37.887,157.150
C00713=1046.255,203.500,-97.318,171.139,37.885,157.150
C00714=1046.249,203.251,-97.293,171.135,37.883,157.149
C00715=1046.243,203.002,-97.268,171.133,37.881,157.149
C00716=1046.237,202.753,-97.242,171.130,37.878,157.148
C00717=1046.230,202.505,-97.217,171.127,37.877,157.148
C00718=1046.225,202.256,-97.193,171.125,37.874,157.147
C00719=1046.218,202.008,-97.168,171.122,37.873,157.147
C00720=1046.212,201.759,-97.143,171.119,37.870,157.146
C00721=1046.206,201.510,-97.118,171.117,37.868,157.146
C00722=1046.200,201.261,-97.093,171.114,37.866,157.146
C00723=1046.195,201.013,-97.068,171.111,37.864,157.145
C00724=1046.188,200.764,-97.044,171.109,37.862,157.145
C00725=1046.182,200.516,-97.018,171.105,37.860,157.144
C00726=1046.175,200.267,-96.994,171.103,37.859,157.144
C00727=1046.169,200.018,-96.969,171.101,37.856,157.143
C00728=1046.163,199.769,-96.945,171.097,37.854,157.143
C00729=1046.157,199.521,-96.920,171.095,37.853,157.142
C00730=1046.151,199.272,-96.895,171.093,37.850,157.142
C00731=1046.144,199.023,-96.871,171.089,37.849,157.142
C00732=1046.138,198.774,-96.846,171.087,37.847,157.141
C00733=1046.132,198.526,-96.821,171.085,37.845,157.141
C00734=1046.126,198.277,-96.797,171.081,37.843,157.140
C00735=1046.120,198.028,-96.772,171.079,37.841,157.140
C00736=1046.113,197.779,-96.748,171.077,37.839,157.139
C00737=1046.107,197.531,-96.723,171.073,37.837,157.139
C00738=1046.100,197.282,-96.699,171.071,37.835,157.139
C00739=1046.095,197.033,-96.674,171.069,37.833,157.138
C00740=1046.089,196.785,-96.649,171.066,37.831,157.138
C00741=1046.082,196.536,-96.625,171.063,37.829,157.137
C00742=1046.076,196.287,-96.600,171.061,37.827,157.137
C00743=1046.069,196.039,-96.576,171.058,37.826,157.136
C00744=1046.064,195.790,-96.551,171.055,37.823,157.136
C00745=1046.058,195.541,-96.527,171.052,37.821,157.136
C00746=1046.051,195.292,-96.502,171.050,37.820,157.135
C00747=1046.046,195.044,-96.478,171.047,37.817,157.135
C00748=1046.039,194.795,-96.454,171.044,37.816,157.134
C00749=1046.033,194.546,-96.428,171.042,37.814,157.134
C00750=1046.027,194.298,-96.405,171.040,37.812,157.133
C00751=1046.021,194.049,-96.380,171.036,37.810,157.133
C00752=1046.015,193.800,-96.356,171.034,37.808,157.133
C00753=1046.009,193.552,-96.331,171.032,37.806,157.132
C00754=1046.002,193.303,-96.307,171.030,37.804,157.132
C00755=1045.997,193.054,-96.283,171.026,37.802,157.131
C00756=1045.990,192.805,-96.259,171.024,37.800,157.131
C00757=1045.984,192.556,-96.233,171.022,37.799,157.130
C00758=1045.979,192.308,-96.209,171.019,37.797,157.130
C00759=1045.972,192.059,-96.185,171.016,37.794,157.129
C00760=1045.967,191.810,-96.161,171.014,37.793,157.129
C00761=1045.960,191.561,-96.137,171.011,37.791,157.129
C00762=1045.954,191.312,-96.112,171.009,37.789,157.128
C00763=1045.948,191.064,-96.088,171.006,37.787,157.128
C00764=1045.942,190.815,-96.063,171.003,37.785,157.127
C00765=1045.936,190.567,-96.040,171.001,37.783,157.127
C00766=1045.930,190.317,-96.015,170.999,37.781,157.127
C00767=1045.924,190.033,-95.988,170.995,37.779,157.126
C00768=1045.916,189.749,-95.960,170.993,37.777,157.126
C00769=1045.909,189.464,-95.932,170.989,37.775,157.125
C00770=1045.903,189.180,-95.904,170.987,37.773,157.125
C00771=1045.897,188.931,-95.880,170.984,37.771,157.124
C00772=1045.891,188.682,-95.856,170.981,37.769,157.124
C00773=1045.885,188.434,-95.832,170.979,37.767,157.123
C00774=1045.879,188.185,-95.807,170.977,37.765,157.123
C00775=1045.873,187.936,-95.784,170.974,37.763,157.123
C00776=1045.867,187.687,-95.759,170.971,37.761,157.122
C00777=1045.861,187.439,-95.735,170.969,37.760,157.122
C00778=1045.854,187.190,-95.711,170.967,37.758,157.121
C00779=1045.849,186.941,-95.687,170.964,37.756,157.121
C00780=1045.843,186.693,-95.663,170.962,37.754,157.120
C00781=1045.837,186.444,-95.639,170.959,37.752,157.120
C00782=1045.831,186.195,-95.615,170.956,37.750,157.120
C00783=1045.825,185.946,-95.590,170.954,37.748,157.119
C00784=1045.819,185.698,-95.567,170.952,37.747,157.119
C00785=1045.814,185.448,-95.543,170.949,37.745,157.119
C00786=1045.807,185.200,-95.519,170.947,37.742,157.118
C00787=1045.802,184.951,-95.495,170.944,37.741,157.118
C00788=1045.796,184.702,-95.471,170.941,37.739,157.117
C00789=1045.790,184.453,-95.447,170.939,37.737,157.117
C00790=1045.784,184.204,-95.423,170.937,37.735,157.116
C00791=1045.778,183.956,-95.398,170.934,37.734,157.116
C00792=1045.772,183.706,-95.375,170.932,37.732,157.116
C00793=1045.766,183.458,-95.351,170.929,37.730,157.115
C00794=1045.759,183.209,-95.327,170.927,37.728,157.115
C00795=1045.753,182.961,-95.304,170.924,37.726,157.115
C00796=1045.747,182.711,-95.280,170.922,37.725,157.114
C00797=1045.741,182.463,-95.257,170.920,37.723,157.114
C00798=1045.734,182.214,-95.233,170.916,37.721,157.113
C00799=1045.728,181.965,-95.210,170.914,37.720,157.113
C00800=1045.722,181.717,-95.187,170.912,37.718,157.113
C00801=1045.715,181.468,-95.163,170.910,37.716,157.112
C00802=1045.709,181.219,-95.140,170.907,37.715,157.112
C00803=1045.703,180.970,-95.116,170.904,37.713,157.112
C00804=1045.697,180.721,-95.093,170.902,37.711,157.111
C00805=1045.690,180.472,-95.069,170.899,37.709,157.111
C00806=1045.684,180.224,-95.045,170.897,37.708,157.110
C00807=1045.678,179.974,-95.022,170.895,37.706,157.110
C00808=1045.672,179.726,-94.998,170.893,37.705,157.110
C00809=1045.666,179.477,-94.975,170.889,37.703,157.109
C00810=1045.660,179.228,-94.951,170.887,37.701,157.109
C00811=1045.654,178.979,-94.928,170.885,37.699,157.109
C00812=1045.647,178.730,-94.904,170.882,37.698,157.108
C00813=1045.641,178.482,-94.882,170.880,37.696,157.108
C00814=1045.635,178.234,-94.858,170.878,37.695,157.107
C00815=1045.628,177.984,-94.835,170.876,37.693,157.107
C00816=1045.622,177.736,-94.811,170.872,37.691,157.107
C00817=1045.616,177.486,-94.788,170.870,37.689,157.106
C00818=1045.610,177.238,-94.764,170.868,37.688,157.106
C00819=1045.604,176.989,-94.741,170.866,37.686,157.106
C00820=1045.598,176.740,-94.717,170.863,37.684,157.105
C00821=1045.592,176.491,-94.694,170.861,37.683,157.105
C00822=1045.586,176.243,-94.671,170.859,37.681,157.104
C00823=1045.579,175.993,-94.648,170.856,37.680,157.104
C00824=1045.573,175.745,-94.625,170.853,37.678,157.104
C00825=1045.567,175.496,-94.601,170.851,37.676,157.103
C00826=1045.561,175.247,-94.578,170.849,37.674,157.103
C00827=1045.555,174.998,-94.554,170.846,37.673,157.103
C00828=1045.549,174.749,-94.531,170.844,37.671,157.102
C00829=1045.543,174.500,-94.508,170.842,37.670,157.102
C00830=1045.537,174.252,-94.484,170.839,37.668,157.102
C00831=1045.530,173.967,-94.459,170.836,37.666,157.101
C00832=1045.523,173.682,-94.431,170.834,37.664,157.101
C00833=1045.515,173.397,-94.405,170.831,37.662,157.100
C00834=1045.509,173.112,-94.379,170.828,37.660,157.100
C00835=1045.502,172.863,-94.355,170.826,37.658,157.100
C00836=1045.497,172.614,-94.332,170.824,37.657,157.099
C00837=1045.490,172.366,-94.310,170.821,37.655,157.099
C00838=1045.484,172.117,-94.287,170.819,37.654,157.099
C00839=1045.478,171.868,-94.263,170.817,37.652,157.098
C00840=1045.472,171.619,-94.240,170.815,37.650,157.098
C00841=1045.466,171.370,-94.217,170.812,37.649,157.097
C00842=1045.461,171.121,-94.194,170.810,37.647,157.097
C00843=1045.454,170.872,-94.170,170.807,37.645,157.097
C00844=1045.447,170.624,-94.148,170.804,37.644,157.096
C00845=1045.442,170.375,-94.125,170.802,37.642,157.096
C00846=1045.436,170.126,-94.102,170.800,37.641,157.096
C00847=1045.430,169.877,-94.079,170.798,37.639,157.095
C00848=1045.424,169.629,-94.055,170.795,37.637,157.095
C00849=1045.418,169.379,-94.032,170.793,37.635,157.095
C00850=1045.411,169.131,-94.009,170.791,37.634,157.094
C00851=1045.406,168.882,-93.986,170.789,37.632,157.094
C00852=1045.400,168.633,-93.963,170.786,37.630,157.093
C00853=1045.394,168.384,-93.941,170.784,37.629,157.093
C00854=1045.389,168.135,-93.918,170.782,37.627,157.093
C00855=1045.382,167.886,-93.894,170.780,37.626,157.092
C00856=1045.375,167.637,-93.871,170.777,37.624,157.092
C00857=1045.370,167.389,-93.848,170.775,37.622,157.092
C00858=1045.364,167.140,-93.825,170.773,37.620,157.091
C00859=1045.358,166.891,-93.802,170.770,37.619,157.091
C00860=1045.352,166.642,-93.779,170.768,37.617,157.091
C00861=1045.347,166.393,-93.756,170.766,37.616,157.090
C00862=1045.340,166.144,-93.734,170.764,37.614,157.090
C00863=1045.335,165.896,-93.711,170.761,37.612,157.089
C00864=1045.328,165.646,-93.688,170.759,37.611,157.089
C00865=1045.322,165.397,-93.665,170.757,37.609,157.089
C00866=1045.317,165.148,-93.642,170.755,37.607,157.088
C00867=1045.310,164.900,-93.620,170.752,37.605,157.088
C00868=1045.305,164.651,-93.597,170.750,37.604,157.088
C00869=1045.299,164.402,-93.574,170.748,37.602,157.087
C00870=1045.293,164.153,-93.551,170.745,37.601,157.087
C00871=1045.287,163.904,-93.528,170.743,37.599,157.087
C00872=1045.281,163.655,-93.505,170.741,37.598,157.086
C00873=1045.275,163.406,-93.483,170.739,37.596,157.086
C00874=1045.269,163.158,-93.460,170.736,37.594,157.086
C00875=1045.264,162.909,-93.437,170.734,37.592,157.085
C00876=1045.257,162.660,-93.414,170.732,37.591,157.085
C00877=1045.252,162.411,-93.391,170.730,37.589,157.085
C00878=1045.246,162.162,-93.368,170.727,37.587,157.084
C00879=1045.240,161.913,-93.346,170.725,37.586,157.084
C00880=1045.235,161.664,-93.323,170.723,37.584,157.083
C00881=1045.228,161.415,-93.301,170.721,37.583,157.083
C00882=1045.222,161.166,-93.278,170.718,37.581,157.083
C00883=1045.217,160.918,-93.255,170.716,37.579,157.082
C00884=1045.211,160.669,-93.232,170.714,37.577,157.082
C00885=1045.204,160.420,-93.210,170.711,37.576,157.082
C00886=1045.199,160.171,-93.187,170.709,37.574,157.081
C00887=1045.193,159.922,-93.165,170.707,37.573,157.081
C00888=1045.187,159.673,-93.142,170.705,37.571,157.081
C00889=1045.181,159.424,-93.121,170.703,37.570,157.080
C00890=1045.174,159.175,-93.098,170.700,37.568,157.080
C00891=1045.169,158.926,-93.075,170.698,37.567,157.080
C00892=1045.162,158.678,-93.053,170.696,37.565,157.079
C00893=1045.157,158.428,-93.031,170.693,37.564,157.079
C00894=1045.150,158.180,-93.008,170.691,37.562,157.079
C00895=1045.143,157.894,-92.983,170.689,37.561,157.078
C00896=1045.135,157.609,-92.957,170.687,37.559,157.078
C00897=1045.129,157.324,-92.932,170.683,37.557,157.078
C00898=1045.122,157.038,-92.905,170.681,37.555,157.077
C00899=1045.116,156.789,-92.884,170.679,37.554,157.077
C00900=1045.110,156.540,-92.861,170.677,37.552,157.077
C00901=1045.104,156.291,-92.839,170.674,37.551,157.076
C00902=1045.098,156.042,-92.817,170.672,37.549,157.076
C00903=1045.091,155.794,-92.794,170.670,37.547,157.076
C00904=1045.086,155.544,-92.772,170.668,37.546,157.075
C00905=1045.079,155.296,-92.750,170.665,37.544,157.075
C00906=1045.074,155.046,-92.728,170.664,37.543,157.075
C00907=1045.067,154.797,-92.705,170.662,37.541,157.074
C00908=1045.061,154.548,-92.684,170.660,37.540,157.074
C00909=1045.055,154.300,-92.661,170.657,37.538,157.074
C00910=1045.049,154.050,-92.639,170.655,37.537,157.073
C00911=1045.043,153.802,-92.617,170.653,37.535,157.073
C00912=1045.037,153.553,-92.595,170.651,37.534,157.073
C00913=1045.031,153.304,-92.573,170.649,37.532,157.072
C00914=1045.025,153.055,-92.551,170.646,37.531,157.072
C00915=1045.019,152.806,-92.528,170.644,37.529,157.072
C00916=1045.013,152.557,-92.507,170.642,37.528,157.072
C00917=1045.006,152.309,-92.484,170.640,37.526,157.071
C00918=1045.001,152.059,-92.462,170.637,37.525,157.071
C00919=1044.995,151.810,-92.441,170.635,37.524,157.071
C00920=1044.988,151.561,-92.418,170.633,37.522,157.070
C00921=1044.982,151.312,-92.397,170.631,37.521,157.070
C00922=1044.976,151.063,-92.374,170.628,37.519,157.070
C00923=1044.971,150.815,-92.352,170.626,37.518,157.069
C00924=1044.965,150.565,-92.331,170.625,37.516,157.069
C00925=1044.958,150.317,-92.308,170.623,37.515,157.069
C00926=1044.952,150.068,-92.287,170.620,37.513,157.068
C00927=1044.946,149.818,-92.265,170.618,37.512,157.068
C00928=1044.940,149.570,-92.242,170.616,37.510,157.068
C00929=1044.934,149.320,-92.221,170.614,37.509,157.067
C00930=1044.928,149.071,-92.199,170.612,37.507,157.067
C00931=1044.922,148.823,-92.177,170.609,37.506,157.067
C00932=1044.916,148.574,-92.155,170.607,37.505,157.067
C00933=1044.910,148.325,-92.134,170.605,37.503,157.066
C00934=1044.903,148.076,-92.112,170.603,37.502,157.066
C00935=1044.897,147.827,-92.090,170.600,37.500,157.065
C00936=1044.892,147.578,-92.067,170.599,37.499,157.065
C00937=1044.885,147.328,-92.046,170.597,37.497,157.065
C00938=1044.880,147.080,-92.025,170.595,37.496,157.065
C00939=1044.873,146.831,-92.002,170.593,37.495,157.064
C00940=1044.867,146.582,-91.981,170.590,37.493,157.064
C00941=1044.861,146.333,-91.959,170.588,37.492,157.064
C00942=1044.855,146.084,-91.937,170.586,37.491,157.063
C00943=1044.849,145.834,-91.916,170.584,37.489,157.063
C00944=1044.843,145.585,-91.894,170.581,37.488,157.063
C00945=1044.837,145.337,-91.872,170.579,37.486,157.063
C00946=1044.830,145.088,-91.851,170.577,37.485,157.062
C00947=1044.824,144.839,-91.829,170.576,37.483,157.062
C00948=1044.817,144.590,-91.808,170.574,37.482,157.062
C00949=1044.811,144.341,-91.786,170.571,37.480,157.061
C00950=1044.806,144.092,-91.765,170.569,37.479,157.061
C00951=1044.800,143.843,-91.743,170.567,37.477,157.061
C00952=1044.793,143.594,-91.722,170.565,37.476,157.060
C00953=1044.787,143.345,-91.700,170.562,37.475,157.060
C00954=1044.781,143.095,-91.678,170.560,37.473,157.060
C00955=1044.775,142.848,-91.656,170.558,37.472,157.059
C00956=1044.769,142.598,-91.635,170.557,37.471,157.059
C00957=1044.763,142.349,-91.613,170.555,37.469,157.059
C00958=1044.757,142.100,-91.591,170.552,37.468,157.059
C00959=1044.750,141.814,-91.567,170.550,37.466,157.058
C00960=1044.743,141.529,-91.542,170.548,37.464,157.058
C00961=1044.736,141.243,-91.518,170.545,37.463,157.058
C00962=1044.729,140.957,-91.493,170.542,37.461,157.057
C00963=1044.723,140.709,-91.472,170.540,37.460,157.057
C00964=1044.717,140.460,-91.450,170.539,37.458,157.057
C00965=1044.710,140.211,-91.429,170.537,37.457,157.056
C00966=1044.704,139.962,-91.407,170.534,37.456,157.056
C00967=1044.699,139.713,-91.386,170.532,37.454,157.056
C00968=1044.693,139.464,-91.364,170.530,37.453,157.055
C00969=1044.686,139.215,-91.343,170.528,37.452,157.055
C00970=1044.681,138.965,-91.322,170.526,37.450,157.055
C00971=1044.674,138.717,-91.301,170.523,37.449,157.055
C00972=1044.668,138.467,-91.279,170.522,37.447,157.054
C00973=1044.662,138.218,-91.258,170.520,37.445,157.054
C00974=1044.656,137.970,-91.237,170.518,37.444,157.054
C00975=1044.650,137.720,-91.215,170.516,37.443,157.053
C00976=1044.643,137.472,-91.194,170.513,37.442,157.053
C00977=1044.638,137.222,-91.173,170.511,37.440,157.053
C00978=1044.632,136.973,-91.152,170.509,37.439,157.052
C00979=1044.626,136.724,-91.130,170.508,37.438,157.052
C00980=1044.619,136.475,-91.109,170.505,37.436,157.052
C00981=1044.613,136.227,-91.088,170.503,37.435,157.052
C00982=1044.607,135.977,-91.067,170.501,37.433,157.051
C00983=1044.600,135.728,-91.046,170.499,37.432,157.051
C00984=1044.595,135.479,-91.025,170.497,37.430,157.051
C00985=1044.589,135.230,-91.003,170.494,37.429,157.050
C00986=1044.582,134.981,-90.982,170.493,37.428,157.050
C00987=1044.577,134.732,-90.961,170.491,37.427,157.050
C00988=1044.570,134.483,-90.940,170.489,37.425,157.050
C00989=1044.564,134.234,-90.919,170.487,37.424,157.049
C00990=1044.558,133.985,-90.898,170.484,37.423,157.049
C00991=1044.552,133.736,-90.876,170.482,37.421,157.049
C00992=1044.545,133.487,-90.855,170.481,37.420,157.048
C00993=1044.540,133.238,-90.834,170.479,37.418,157.048
C00994=1044.534,132.989,-90.813,170.477,37.417,157.048
C00995=1044.527,132.740,-90.793,170.474,37.415,157.048
C00996=1044.521,132.491,-90.771,170.472,37.414,157.047
C00997=1044.515,132.241,-90.750,170.470,37.413,157.047
C00998=1044.509,131.993,-90.729,170.469,37.412,157.047
C00999=1044.503,131.744,-90.708,170.466,37.410,157.046
C01000=1044.498,131.495,-90.687,170.464,37.409,157.046
C01001=1044.491,131.246,-90.666,170.462,37.408,157.046
C01002=1044.485,130.996,-90.645,170.460,37.406,157.046
C01003=1044.479,130.748,-90.624,170.459,37.405,157.045
C01004=1044.473,130.498,-90.604,170.456,37.403,157.045
C01005=1044.466,130.249,-90.583,170.454,37.402,157.045
C01006=1044.460,130.000,-90.563,170.452,37.401,157.044
C01007=1044.454,129.751,-90.541,170.450,37.400,157.044
C01008=1044.447,129.502,-90.521,170.448,37.399,157.044
C01009=1044.441,129.253,-90.500,170.446,37.397,157.044
C01010=1044.435,129.004,-90.479,170.444,37.396,157.043
C01011=1044.428,128.755,-90.458,170.442,37.395,157.043
C01012=1044.423,128.506,-90.437,170.440,37.394,157.043
C01013=1044.416,128.257,-90.416,170.438,37.392,157.043
C01014=1044.410,128.008,-90.396,170.436,37.391,157.042
C01015=1044.404,127.759,-90.375,170.433,37.389,157.042
C01016=1044.398,127.510,-90.355,170.432,37.388,157.042
C01017=1044.391,127.261,-90.334,170.430,37.387,157.042
C01018=1044.385,127.011,-90.313,170.428,37.386,157.041
C01019=1044.379,126.762,-90.293,170.426,37.385,157.041
C01020=1044.372,126.513,-90.272,170.423,37.383,157.041
C01021=1044.367,126.264,-90.251,170.422,37.382,157.040
C01022=1044.360,126.015,-90.230,170.420,37.380,157.040
C01023=1044.353,125.729,-90.207,170.418,37.379,157.040
C01024=1044.346,125.443,-90.183,170.416,37.377,157.040
C01025=1044.339,125.158,-90.160,170.412,37.376,157.039
C01026=1044.332,124.872,-90.136,170.410,37.374,157.039
C01027=1044.326,124.623,-90.115,170.409,37.373,157.039
C01028=1044.319,124.373,-90.095,170.407,37.372,157.038
C01029=1044.313,124.125,-90.074,170.405,37.371,157.038
C01030=1044.307,123.875,-90.053,170.402,37.370,157.038
C01031=1044.301,123.626,-90.033,170.400,37.368,157.038
C01032=1044.294,123.377,-90.012,170.399,37.367,157.037
C01033=1044.289,123.128,-89.992,170.397,37.365,157.037
C01034=1044.282,122.879,-89.971,170.395,37.364,157.037
C01035=1044.276,122.631,-89.951,170.392,37.363,157.037
C01036=1044.270,122.381,-89.930,170.390,37.362,157.036
C01037=1044.264,122.132,-89.910,170.389,37.360,157.036
C01038=1044.258,121.883,-89.890,170.387,37.359,157.036
C01039=1044.252,121.634,-89.868,170.385,37.358,157.036
C01040=1044.246,121.385,-89.848,170.382,37.356,157.035
C01041=1044.239,121.136,-89.828,170.381,37.355,157.035
C01042=1044.234,120.886,-89.807,170.379,37.354,157.035
C01043=1044.227,120.638,-89.786,170.377,37.353,157.034
C01044=1044.221,120.389,-89.766,170.375,37.351,157.034
C01045=1044.215,120.139,-89.745,170.372,37.350,157.034
C01046=1044.209,119.890,-89.725,170.371,37.348,157.033
C01047=1044.203,119.641,-89.705,170.369,37.347,157.033
C01048=1044.197,119.392,-89.684,170.367,37.346,157.033
C01049=1044.191,119.143,-89.664,170.365,37.345,157.033
C01050=1044.185,118.894,-89.644,170.363,37.344,157.032
C01051=1044.179,118.645,-89.624,170.361,37.342,157.032
C01052=1044.173,118.395,-89.603,170.359,37.340,157.032
C01053=1044.167,118.146,-89.583,170.357,37.339,157.032
C01054=1044.161,117.898,-89.562,170.356,37.338,157.031
C01055=1044.154,117.649,-89.542,170.353,37.337,157.031
C01056=1044.149,117.400,-89.521,170.351,37.336,157.031
C01057=1044.142,117.150,-89.501,170.349,37.334,157.030
C01058=1044.136,116.901,-89.481,170.347,37.333,157.030
C01059=1044.131,116.652,-89.460,170.346,37.331,157.030
C01060=1044.124,116.403,-89.440,170.343,37.330,157.030
C01061=1044.118,116.154,-89.420,170.341,37.329,157.029
C01062=1044.112,115.905,-89.400,170.339,37.328,157.029
C01063=1044.106,115.655,-89.379,170.338,37.326,157.029
C01064=1044.100,115.407,-89.358,170.336,37.325,157.029
C01065=1044.094,115.158,-89.339,170.333,37.323,157.028
C01066=1044.088,114.908,-89.318,170.332,37.322,157.028
C01067=1044.082,114.659,-89.298,170.330,37.321,157.028
C01068=1044.076,114.411,-89.278,170.328,37.319,157.027
C01069=1044.070,114.161,-89.257,170.326,37.318,157.027
C01070=1044.064,113.912,-89.237,170.324,37.317,157.027
C01071=1044.058,113.663,-89.217,170.322,37.316,157.027
C01072=1044.052,113.414,-89.197,170.320,37.314,157.026
C01073=1044.046,113.165,-89.177,170.318,37.313,157.026
C01074=1044.040,112.916,-89.157,170.317,37.312,157.026
C01075=1044.034,112.666,-89.137,170.315,37.311,157.026
C01076=1044.028,112.417,-89.117,170.312,37.309,157.025
C01077=1044.022,112.168,-89.097,170.310,37.308,157.025
C01078=1044.015,111.919,-89.077,170.309,37.306,157.025
C01079=1044.009,111.670,-89.057,170.307,37.305,157.025
C01080=1044.002,111.420,-89.036,170.305,37.304,157.024
C01081=1043.996,111.172,-89.016,170.302,37.303,157.024
C01082=1043.990,110.923,-88.997,170.301,37.302,157.024
C01083=1043.984,110.674,-88.977,170.299,37.300,157.024
C01084=1043.978,110.424,-88.957,170.297,37.299,157.023
C01085=1043.972,110.175,-88.937,170.295,37.298,157.023
C01086=1043.966,109.926,-88.917,170.293,37.297,157.023
C01087=1043.958,109.640,-88.894,170.290,37.296,157.023
C01088=1043.951,109.354,-88.871,170.288,37.294,157.022
C01089=1043.944,109.068,-88.849,170.286,37.293,157.022
C01090=1043.937,108.782,-88.826,170.284,37.291,157.022
C01091=1043.931,108.533,-88.806,170.283,37.290,157.021
C01092=1043.925,108.284,-88.786,170.280,37.289,157.021
C01093=1043.918,108.035,-88.767,170.278,37.288,157.021
C01094=1043.912,107.786,-88.747,170.276,37.286,157.021
C01095=1043.906,107.536,-88.727,170.275,37.285,157.020
C01096=1043.900,107.288,-88.707,170.273,37.284,157.020
C01097=1043.894,107.038,-88.688,170.270,37.283,157.020
C01098=1043.887,106.789,-88.667,170.268,37.282,157.020
C01099=1043.881,106.540,-88.647,170.267,37.280,157.019
C01100=1043.875,106.291,-88.629,170.265,37.279,157.019
C01101=1043.869,106.042,-88.609,170.263,37.278,157.019
C01102=1043.862,105.792,-88.588,170.261,37.277,157.019
C01103=1043.857,105.543,-88.569,170.259,37.275,157.018
C01104=1043.851,105.294,-88.549,170.257,37.274,157.018
C01105=1043.845,105.045,-88.529,170.255,37.273,157.018
C01106=1043.838,104.795,-88.510,170.253,37.272,157.018
C01107=1043.832,104.547,-88.490,170.252,37.271,157.017
C01108=1043.826,104.298,-88.470,170.249,37.269,157.017
C01109=1043.820,104.048,-88.451,170.247,37.268,157.017
C01110=1043.813,103.799,-88.431,170.246,37.266,157.017
C01111=1043.807,103.550,-88.411,170.244,37.265,157.016
C01112=1043.801,103.301,-88.392,170.242,37.264,157.016
C01113=1043.795,103.052,-88.372,170.240,37.263,157.016
C01114=1043.789,102.803,-88.353,170.238,37.261,157.016
C01115=1043.783,102.553,-88.333,170.236,37.260,157.015
C01116=1043.777,102.304,-88.313,170.234,37.259,157.015
C01117=1043.770,102.055,-88.294,170.232,37.258,157.015
C01118=1043.764,101.806,-88.274,170.231,37.257,157.015
C01119=1043.759,101.557,-88.255,170.229,37.255,157.014
C01120=1043.752,101.307,-88.235,170.226,37.254,157.014
C01121=1043.746,101.058,-88.215,170.225,37.253,157.014
C01122=1043.740,100.810,-88.196,170.223,37.252,157.014
C01123=1043.734,100.560,-88.177,170.221,37.251,157.013
C01124=1043.728,100.311,-88.157,170.219,37.249,157.013
C01125=1043.721,100.062,-88.138,170.217,37.248,157.013
C01126=1043.715,99.813,-88.118,170.215,37.247,157.013
C01127=1043.709,99.563,-88.099,170.213,37.246,157.012
C01128=1043.703,99.314,-88.080,170.211,37.244,157.012
C01129=1043.697,99.065,-88.060,170.210,37.243,157.012
C01130=1043.690,98.816,-88.041,170.208,37.242,157.012
C01131=1043.684,98.567,-88.021,170.205,37.241,157.011
C01132=1043.677,98.317,-88.002,170.204,37.240,157.011
C01133=1043.672,98.068,-87.983,170.202,37.238,157.011
C01134=1043.665,97.820,-87.964,170.200,37.238,157.011
C01135=1043.659,97.570,-87.944,170.198,37.236,157.010
C01136=1043.653,97.321,-87.924,170.197,37.235,157.010
C01137=1043.646,97.071,-87.905,170.194,37.234,157.010
C01138=1043.640,96.822,-87.886,170.192,37.233,157.010
C01139=1043.634,96.574,-87.867,170.190,37.232,157.009
C01140=1043.628,96.324,-87.848,170.189,37.230,157.009
C01141=1043.622,96.075,-87.829,170.187,37.229,157.009
C01142=1043.616,95.826,-87.809,170.185,37.228,157.009
C01143=1043.609,95.577,-87.790,170.182,37.227,157.008
C01144=1043.603,95.327,-87.771,170.181,37.225,157.008
C01145=1043.596,95.078,-87.751,170.179,37.224,157.008
C01146=1043.591,94.829,-87.732,170.177,37.223,157.008
C01147=1043.584,94.580,-87.713,170.176,37.222,157.007
C01148=1043.578,94.330,-87.694,170.174,37.221,157.007
C01149=1043.572,94.082,-87.674,170.171,37.219,157.007
C01150=1043.566,93.833,-87.656,170.169,37.218,157.007
C01151=1043.559,93.546,-87.634,170.167,37.217,157.006
C01152=1043.551,93.260,-87.612,170.166,37.216,157.006
C01153=1043.545,92.974,-87.589,170.164,37.214,157.006
C01154=1043.538,92.688,-87.567,170.161,37.213,157.006
C01155=1043.531,92.439,-87.548,170.159,37.211,157.005
C01156=1043.525,92.190,-87.529,170.157,37.210,157.005
C01157=1043.519,91.940,-87.511,170.155,37.209,157.005
C01158=1043.513,91.692,-87.491,170.154,37.208,157.005
C01159=1043.507,91.443,-87.472,170.152,37.207,157.004
C01160=1043.501,91.193,-87.453,170.149,37.205,157.004
C01161=1043.495,90.944,-87.434,170.148,37.204,157.004
C01162=1043.489,90.695,-87.415,170.146,37.203,157.004
C01163=1043.482,90.446,-87.395,170.144,37.202,157.003
C01164=1043.476,90.197,-87.376,170.143,37.200,157.003
C01165=1043.470,89.947,-87.358,170.141,37.200,157.003
C01166=1043.464,89.698,-87.339,170.138,37.199,157.003
C01167=1043.457,89.449,-87.320,170.136,37.197,157.002
C01168=1043.451,89.200,-87.301,170.135,37.196,157.002
C01169=1043.444,88.950,-87.282,170.133,37.195,157.002
C01170=1043.438,88.701,-87.263,170.131,37.194,157.002
C01171=1043.432,88.452,-87.245,170.129,37.193,157.002
C01172=1043.426,88.202,-87.225,170.127,37.192,157.001
C01173=1043.419,87.953,-87.207,170.125,37.191,157.001
C01174=1043.413,87.704,-87.188,170.123,37.189,157.001
C01175=1043.407,87.455,-87.170,170.122,37.188,157.001
C01176=1043.401,87.206,-87.150,170.120,37.187,157.000
C01177=1043.394,86.956,-87.132,170.118,37.186,157.000
C01178=1043.388,86.707,-87.113,170.115,37.185,157.000
C01179=1043.382,86.458,-87.094,170.114,37.184,157.000
C01180=1043.376,86.209,-87.075,170.112,37.183,156.999
C01181=1043.370,85.960,-87.056,170.110,37.181,156.999
C01182=1043.363,85.710,-87.038,170.108,37.180,156.999
C01183=1043.357,85.461,-87.019,170.107,37.179,156.999
C01184=1043.351,85.212,-87.000,170.104,37.178,156.998
C01185=1043.345,84.963,-86.981,170.102,37.177,156.998
C01186=1043.338,84.714,-86.963,170.101,37.176,156.998
C01187=1043.332,84.465,-86.944,170.099,37.175,156.998
C01188=1043.325,84.215,-86.925,170.097,37.174,156.998
C01189=1043.320,83.966,-86.906,170.095,37.172,156.997
C01190=1043.313,83.717,-86.887,170.094,37.171,156.997
C01191=1043.307,83.468,-86.869,170.091,37.170,156.997
C01192=1043.301,83.218,-86.851,170.089,37.169,156.997
C01193=1043.294,82.969,-86.832,170.088,37.167,156.996
C01194=1043.288,82.719,-86.813,170.086,37.166,156.996
C01195=1043.282,82.470,-86.794,170.084,37.166,156.996
C01196=1043.276,82.222,-86.776,170.083,37.164,156.996
C01197=1043.270,81.973,-86.757,170.080,37.163,156.996
C01198=1043.264,81.723,-86.738,170.078,37.162,156.995
C01199=1043.258,81.474,-86.720,170.076,37.161,156.995
C01200=1043.252,81.224,-86.702,170.075,37.159,156.995
C01201=1043.245,80.975,-86.683,170.073,37.158,156.995
C01202=1043.239,80.726,-86.664,170.071,37.157,156.994
C01203=1043.232,80.477,-86.646,170.069,37.156,156.994
C01204=1043.227,80.228,-86.626,170.067,37.154,156.994
C01205=1043.220,79.978,-86.608,170.065,37.154,156.994
C01206=1043.214,79.729,-86.590,170.063,37.153,156.993
C01207=1043.208,79.480,-86.571,170.062,37.151,156.993
C01208=1043.202,79.231,-86.553,170.060,37.150,156.993
C01209=1043.196,78.982,-86.534,170.057,37.149,156.993
C01210=1043.190,78.732,-86.516,170.056,37.148,156.992
C01211=1043.184,78.483,-86.497,170.054,37.147,156.992
C01212=1043.177,78.234,-86.478,170.052,37.145,156.992
C01213=1043.171,77.984,-86.460,170.051,37.144,156.992
C01214=1043.165,77.735,-86.442,170.049,37.143,156.991
C01215=1043.158,77.449,-86.421,170.046,37.142,156.991
C01216=1043.150,77.163,-86.399,170.044,37.140,156.991
C01217=1043.143,76.877,-86.378,170.042,37.139,156.991
C01218=1043.136,76.591,-86.358,170.040,37.138,156.990
C01219=1043.130,76.342,-86.339,170.038,37.137,156.990
C01220=1043.123,76.093,-86.321,170.037,37.135,156.990
C01221=1043.117,75.843,-86.303,170.034,37.135,156.990
C01222=1043.111,75.594,-86.284,170.032,37.134,156.990
C01223=1043.105,75.344,-86.266,170.030,37.132,156.989
C01224=1043.099,75.096,-86.248,170.029,37.131,156.989
C01225=1043.092,74.847,-86.229,170.027,37.130,156.989
C01226=1043.086,74.597,-86.211,170.025,37.129,156.989
C01227=1043.080,74.348,-86.193,170.024,37.128,156.988
C01228=1043.074,74.098,-86.175,170.021,37.127,156.988
C01229=1043.067,73.849,-86.156,170.019,37.126,156.988
C01230=1043.061,73.600,-86.137,170.017,37.124,156.988
C01231=1043.055,73.351,-86.120,170.016,37.124,156.988
C01232=1043.048,73.102,-86.102,170.014,37.123,156.987
C01233=1043.042,72.852,-86.084,170.012,37.121,156.987
C01234=1043.036,72.603,-86.065,170.010,37.120,156.987
C01235=1043.029,72.353,-86.047,170.008,37.119,156.987
C01236=1043.024,72.105,-86.029,170.006,37.118,156.986
C01237=1043.018,71.855,-86.011,170.004,37.117,156.986
C01238=1043.011,71.606,-85.992,170.003,37.116,156.986
C01239=1043.005,71.356,-85.974,170.001,37.115,156.986
C01240=1042.999,71.107,-85.956,169.999,37.113,156.986
C01241=1042.992,70.859,-85.939,169.997,37.112,156.985
C01242=1042.986,70.609,-85.920,169.995,37.111,156.985
C01243=1042.980,70.360,-85.902,169.993,37.110,156.985
C01244=1042.973,70.111,-85.884,169.991,37.109,156.985
C01245=1042.967,69.861,-85.866,169.990,37.108,156.984
C01246=1042.962,69.612,-85.848,169.988,37.107,156.984
C01247=1042.955,69.363,-85.829,169.985,37.105,156.984
C01248=1042.948,69.113,-85.812,169.984,37.105,156.984
C01249=1042.942,68.864,-85.793,169.982,37.103,156.984
C01250=1042.936,68.615,-85.776,169.980,37.102,156.983
C01251=1042.930,68.365,-85.758,169.978,37.101,156.983
C01252=1042.923,68.117,-85.740,169.977,37.100,156.983
C01253=1042.917,67.867,-85.722,169.975,37.099,156.983
C01254=1042.911,67.617,-85.704,169.972,37.098,156.982
C01255=1042.905,67.369,-85.686,169.971,37.097,156.982
C01256=1042.898,67.119,-85.668,169.969,37.095,156.982
C01257=1042.892,66.869,-85.650,169.967,37.095,156.982
C01258=1042.886,66.620,-85.632,169.965,37.094,156.982
C01259=1042.880,66.371,-85.614,169.964,37.092,156.981
C01260=1042.873,66.122,-85.597,169.961,37.091,156.981
C01261=1042.867,65.873,-85.578,169.959,37.091,156.981
C01262=1042.861,65.624,-85.561,169.957,37.089,156.981
C01263=1042.855,65.374,-85.543,169.956,37.088,156.980
C01264=1042.848,65.125,-85.525,169.954,37.087,156.980
C01265=1042.842,64.875,-85.507,169.952,37.086,156.980
C01266=1042.836,64.627,-85.490,169.951,37.085,156.980
C01267=1042.830,64.377,-85.472,169.948,37.084,156.980
C01268=1042.823,64.127,-85.454,169.946,37.083,156.979
C01269=1042.816,63.878,-85.436,169.944,37.081,156.979
C01270=1042.811,63.629,-85.418,169.943,37.081,156.979
C01271=1042.804,63.380,-85.401,169.941,37.079,156.979
C01272=1042.798,63.130,-85.383,169.939,37.079,156.979
C01273=1042.791,62.881,-85.366,169.937,37.078,156.978
C01274=1042.785,62.632,-85.348,169.935,37.076,156.978
C01275=1042.778,62.383,-85.330,169.933,37.076,156.978
C01276=1042.771,62.133,-85.313,169.931,37.075,156.978
C01277=1042.765,61.884,-85.295,169.929,37.073,156.978
C01278=1042.759,61.635,-85.278,169.928,37.073,156.977
C01279=1042.751,61.348,-85.258,169.926,37.071,156.977
C01280=1042.745,61.062,-85.238,169.924,37.070,156.977
C01281=1042.737,60.776,-85.217,169.921,37.069,156.977
C01282=1042.730,60.490,-85.197,169.919,37.068,156.976
C01283=1042.723,60.240,-85.180,169.917,37.067,156.976
C01284=1042.717,59.991,-85.162,169.915,37.066,156.976
C01285=1042.711,59.742,-85.145,169.913,37.065,156.976
C01286=1042.705,59.492,-85.127,169.912,37.064,156.976
C01287=1042.698,59.243,-85.110,169.910,37.063,156.975
C01288=1042.691,58.994,-85.092,169.907,37.062,156.975
C01289=1042.685,58.745,-85.074,169.905,37.061,156.975
C01290=1042.678,58.495,-85.057,169.904,37.060,156.975
C01291=1042.672,58.246,-85.039,169.902,37.059,156.975
C01292=1042.666,57.997,-85.022,169.900,37.058,156.974
C01293=1042.659,57.748,-85.005,169.898,37.057,156.974
C01294=1042.653,57.499,-84.987,169.897,37.055,156.974
C01295=1042.647,57.249,-84.970,169.895,37.055,156.974
C01296=1042.640,56.999,-84.952,169.892,37.054,156.974
C01297=1042.634,56.751,-84.935,169.890,37.052,156.973
C01298=1042.628,56.501,-84.918,169.889,37.052,156.973
C01299=1042.622,56.251,-84.900,169.887,37.050,156.973
C01300=1042.615,56.002,-84.883,169.885,37.049,156.973
C01301=1042.609,55.752,-84.865,169.883,37.049,156.973
C01302=1042.603,55.504,-84.848,169.882,37.047,156.972
C01303=1042.596,55.254,-84.831,169.879,37.046,156.972
C01304=1042.590,55.004,-84.813,169.877,37.046,156.972
C01305=1042.584,54.756,-84.796,169.875,37.044,156.972
C01306=1042.577,54.506,-84.779,169.874,37.043,156.971
C01307=1042.571,54.257,-84.761,169.872,37.042,156.971
C01308=1042.564,54.008,-84.744,169.870,37.041,156.971
C01309=1042.558,53.758,-84.726,169.868,37.040,156.971
C01310=1042.552,53.509,-84.710,169.866,37.039,156.971
C01311=1042.546,53.259,-84.692,169.864,37.038,156.971
C01312=1042.540,53.010,-84.675,169.862,37.037,156.970
C01313=1042.533,52.761,-84.657,169.861,37.036,156.970
C01314=1042.527,52.512,-84.640,169.859,37.035,156.970
C01315=1042.521,52.262,-84.623,169.857,37.034,156.970
C01316=1042.515,52.014,-84.606,169.855,37.033,156.969
C01317=1042.508,51.764,-84.589,169.853,37.032,156.969
C01318=1042.502,51.514,-84.571,169.851,37.031,156.969
C01319=1042.496,51.265,-84.554,169.849,37.029,156.969
C01320=1042.489,51.015,-84.536,169.847,37.028,156.969
C01321=1042.483,50.767,-84.519,169.846,37.028,156.968
C01322=1042.477,50.517,-84.502,169.844,37.026,156.968
C01323=1042.471,50.268,-84.485,169.842,37.025,156.968
C01324=1042.464,50.018,-84.468,169.840,37.025,156.968
C01325=1042.458,49.769,-84.451,169.838,37.023,156.968
C01326=1042.452,49.519,-84.433,169.836,37.022,156.967
C01327=1042.446,49.270,-84.416,169.834,37.021,156.967
C01328=1042.439,49.021,-84.399,169.832,37.020,156.967
C01329=1042.434,48.772,-84.382,169.831,37.019,156.967
C01330=1042.427,48.522,-84.365,169.829,37.018,156.966
C01331=1042.421,48.273,-84.348,169.827,37.017,156.966
C01332=1042.415,48.024,-84.330,169.824,37.016,156.966
C01333=1042.408,47.775,-84.313,169.823,37.015,156.966
C01334=1042.402,47.525,-84.297,169.821,37.013,156.966
C01335=1042.396,47.276,-84.279,169.819,37.013,156.965
C01336=1042.390,47.027,-84.262,169.818,37.012,156.965
C01337=1042.384,46.777,-84.245,169.816,37.010,156.965
C01338=1042.378,46.528,-84.228,169.813,37.009,156.965
C01339=1042.371,46.278,-84.210,169.811,37.008,156.965
C01340=1042.365,46.029,-84.194,169.810,37.007,156.964
C01341=1042.360,45.780,-84.176,169.808,37.006,156.964
C01342=1042.353,45.530,-84.159,169.806,37.005,156.964
C01343=1042.346,45.244,-84.140,169.804,37.003,156.964
C01344=1042.339,44.957,-84.120,169.802,37.002,156.963
C01345=1042.332,44.671,-84.100,169.799,37.001,156.963
C01346=1042.325,44.384,-84.082,169.797,37.000,156.963
C01347=1042.318,44.135,-84.064,169.795,36.999,156.963
C01348=1042.312,43.885,-84.048,169.794,36.998,156.963
C01349=1042.306,43.637,-84.031,169.792,36.997,156.962
C01350=1042.300,43.386,-84.013,169.790,36.995,156.962
C01351=1042.294,43.138,-83.996,169.788,36.995,156.962
C01352=1042.287,42.888,-83.979,169.786,36.994,156.962
C01353=1042.281,42.639,-83.963,169.784,36.993,156.962
C01354=1042.274,42.389,-83.945,169.782,36.992,156.961
C01355=1042.269,42.140,-83.929,169.780,36.990,156.961
C01356=1042.263,41.891,-83.913,169.779,36.990,156.961
C01357=1042.256,41.641,-83.896,169.777,36.989,156.961
C01358=1042.250,41.392,-83.879,169.775,36.987,156.961
C01359=1042.243,41.142,-83.862,169.773,36.987,156.960
C01360=1042.237,40.893,-83.846,169.770,36.985,156.960
C01361=1042.231,40.644,-83.829,169.769,36.985,156.960
C01362=1042.224,40.394,-83.812,169.767,36.984,156.960
C01363=1042.218,40.146,-83.795,169.765,36.982,156.960
C01364=1042.212,39.896,-83.779,169.763,36.982,156.959
C01365=1042.206,39.646,-83.761,169.762,36.980,156.959
C01366=1042.200,39.397,-83.745,169.760,36.979,156.959
C01367=1042.193,39.147,-83.728,169.757,36.979,156.959
C01368=1042.187,38.898,-83.711,169.755,36.977,156.959
C01369=1042.181,38.649,-83.695,169.754,36.977,156.958
C01370=1042.174,38.400,-83.678,169.752,36.976,156.958
C01371=1042.168,38.150,-83.661,169.750,36.974,156.958
C01372=1042.162,37.901,-83.645,169.748,36.974,156.958
C01373=1042.155,37.651,-83.628,169.746,36.972,156.958
C01374=1042.150,37.402,-83.611,169.745,36.971,156.957
C01375=1042.144,37.153,-83.595,169.742,36.971,156.957
C01376=1042.137,36.903,-83.579,169.740,36.969,156.957
C01377=1042.130,36.654,-83.562,169.738,36.969,156.957
C01378=1042.124,36.405,-83.546,169.736,36.967,156.957
C01379=1042.118,36.155,-83.529,169.735,36.967,156.956
C01380=1042.111,35.906,-83.512,169.733,36.966,156.956
C01381=1042.105,35.656,-83.496,169.731,36.965,156.956
C01382=1042.099,35.407,-83.479,169.729,36.964,156.956
C01383=1042.092,35.158,-83.464,169.726,36.963,156.956
C01384=1042.085,34.908,-83.446,169.725,36.962,156.956
C01385=1042.079,34.659,-83.430,169.723,36.961,156.955
C01386=1042.073,34.410,-83.414,169.721,36.960,156.955
C01387=1042.067,34.160,-83.398,169.719,36.959,156.955
C01388=1042.060,33.910,-83.382,169.717,36.958,156.955
C01389=1042.054,33.662,-83.365,169.716,36.957,156.955
C01390=1042.048,33.412,-83.348,169.714,36.956,156.954
C01391=1042.041,33.162,-83.332,169.711,36.955,156.954
C01392=1042.035,32.913,-83.316,169.709,36.954,156.954
C01393=1042.029,32.664,-83.300,169.707,36.953,156.954
C01394=1042.022,32.415,-83.283,169.706,36.953,156.954
C01395=1042.016,32.165,-83.266,169.704,36.951,156.953
C01396=1042.010,31.916,-83.250,169.702,36.951,156.953
C01397=1042.004,31.667,-83.234,169.700,36.949,156.953
C01398=1041.997,31.417,-83.218,169.698,36.949,156.953
C01399=1041.991,31.167,-83.201,169.696,36.948,156.953
C01400=1041.985,30.918,-83.185,169.694,36.946,156.952
C01401=1041.979,30.669,-83.169,169.692,36.946,156.952
C01402=1041.972,30.419,-83.152,169.690,36.944,156.952
C01403=1041.965,30.170,-83.136,169.688,36.944,156.952
C01404=1041.959,29.921,-83.120,169.687,36.943,156.952
C01405=1041.953,29.672,-83.103,169.685,36.942,156.952
C01406=1041.947,29.422,-83.087,169.683,36.941,156.951
C01407=1041.939,29.135,-83.068,169.680,36.939,156.951
C01408=1041.932,28.848,-83.050,169.678,36.938,156.951
C01409=1041.926,28.562,-83.031,169.676,36.938,156.951
C01410=1041.918,28.276,-83.012,169.674,36.936,156.951
C01411=1041.912,28.026,-82.996,169.672,36.935,156.950
C01412=1041.905,27.776,-82.980,169.670,36.935,156.950
C01413=1041.899,27.527,-82.964,169.668,36.934,156.950
C01414=1041.892,27.278,-82.948,169.666,36.933,156.950
C01415=1041.886,27.029,-82.932,169.664,36.932,156.950
C01416=1041.880,26.779,-82.915,169.662,36.931,156.949
C01417=1041.873,26.530,-82.900,169.660,36.930,156.949
C01418=1041.868,26.280,-82.884,169.658,36.929,156.949
C01419=1041.861,26.031,-82.868,169.656,36.928,156.949
C01420=1041.855,25.781,-82.852,169.654,36.927,156.949
C01421=1041.848,25.531,-82.836,169.653,36.926,156.949
C01422=1041.842,25.282,-82.820,169.651,36.925,156.948
C01423=1041.836,25.033,-82.804,169.648,36.925,156.948
C01424=1041.829,24.784,-82.788,169.646,36.923,156.948
C01425=1041.823,24.535,-82.772,169.644,36.923,156.948
C01426=1041.816,24.285,-82.756,169.642,36.922,156.948
C01427=1041.810,24.035,-82.739,169.641,36.921,156.948
C01428=1041.804,23.785,-82.724,169.639,36.920,156.947
C01429=1041.798,23.536,-82.708,169.637,36.919,156.947
C01430=1041.792,23.287,-82.692,169.635,36.918,156.947
C01431=1041.785,23.038,-82.676,169.633,36.917,156.947
C01432=1041.779,22.789,-82.660,169.630,36.916,156.947
C01433=1041.772,22.539,-82.644,169.628,36.915,156.946
C01434=1041.766,22.289,-82.628,169.627,36.915,156.946
C01435=1041.759,22.040,-82.613,169.625,36.913,156.946
C01436=1041.753,21.791,-82.597,169.623,36.913,156.946
C01437=1041.747,21.542,-82.581,169.621,36.911,156.946
C01438=1041.741,21.292,-82.565,169.619,36.911,156.946
C01439=1041.735,21.042,-82.549,169.617,36.910,156.945
C01440=1041.728,20.793,-82.533,169.616,36.909,156.945
C01441=1041.722,20.544,-82.517,169.613,36.908,156.945
C01442=1041.715,20.294,-82.501,169.611,36.907,156.945
C01443=1041.709,20.044,-82.486,169.609,36.907,156.945
C01444=1041.703,19.795,-82.470,169.607,36.905,156.944
C01445=1041.697,19.546,-82.454,169.605,36.905,156.944
C01446=1041.690,19.297,-82.438,169.603,36.903,156.944
C01447=1041.684,19.047,-82.423,169.602,36.903,156.944
C01448=1041.678,18.798,-82.407,169.600,36.902,156.944
C01449=1041.671,18.549,-82.391,169.597,36.901,156.944
C01450=1041.665,18.299,-82.376,169.595,36.900,156.944
C01451=1041.659,18.050,-82.360,169.593,36.899,156.943
C01452=1041.652,17.800,-82.344,169.591,36.898,156.943
C01453=1041.646,17.550,-82.328,169.589,36.898,156.943
C01454=1041.639,17.301,-82.313,169.588,36.897,156.943
C01455=1041.633,17.052,-82.296,169.586,36.896,156.943
C01456=1041.627,16.802,-82.282,169.584,36.895,156.942
C01457=1041.620,16.553,-82.266,169.582,36.894,156.942
C01458=1041.615,16.303,-82.250,169.579,36.893,156.942
C01459=1041.608,16.054,-82.235,169.577,36.892,156.942
C01460=1041.601,15.805,-82.219,169.575,36.892,156.942
C01461=1041.595,15.555,-82.203,169.573,36.890,156.942
C01462=1041.589,15.306,-82.188,169.572,36.890,156.941
C01463=1041.583,15.056,-82.172,169.570,36.888,156.941
C01464=1041.576,14.807,-82.157,169.568,36.888,156.941
C01465=1041.570,14.558,-82.141,169.566,36.887,156.941
C01466=1041.564,14.308,-82.125,169.564,36.886,156.941
C01467=1041.557,14.059,-82.110,169.561,36.885,156.941
C01468=1041.551,13.809,-82.095,169.559,36.884,156.940
C01469=1041.544,13.560,-82.079,169.557,36.883,156.940
C01470=1041.539,13.310,-82.064,169.555,36.883,156.940
C01471=1041.531,13.025,-82.046,169.553,36.882,156.940
C01472=1041.524,12.740,-82.028,169.551,36.881,156.940
C01473=1041.516,12.454,-82.011,169.549,36.880,156.940
C01474=1041.509,12.169,-81.994,169.547,36.879,156.939
C01475=1041.502,11.920,-81.978,169.545,36.878,156.939
C01476=1041.496,11.670,-81.963,169.543,36.878,156.939
C01477=1041.489,11.420,-81.948,169.540,36.877,156.939
C01478=1041.483,11.171,-81.932,169.538,36.876,156.939
C01479=1041.477,10.921,-81.917,169.536,36.875,156.939
C01480=1041.470,10.672,-81.901,169.534,36.874,156.938
C01481=1041.464,10.423,-81.886,169.532,36.873,156.938
C01482=1041.458,10.173,-81.871,169.530,36.873,156.938
C01483=1041.451,9.924,-81.856,169.528,36.872,156.938
C01484=1041.445,9.674,-81.841,169.527,36.871,156.938
C01485=1041.438,9.425,-81.825,169.525,36.870,156.938
C01486=1041.431,9.176,-81.810,169.523,36.870,156.938
C01487=1041.426,8.926,-81.795,169.520,36.869,156.937
C01488=1041.419,8.677,-81.779,169.518,36.868,156.937
C01489=1041.413,8.427,-81.764,169.516,36.867,156.937
C01490=1041.406,8.177,-81.749,169.514,36.867,156.937
C01491=1041.400,7.928,-81.733,169.512,36.865,156.937
C01492=1041.393,7.679,-81.718,169.510,36.865,156.937
C01493=1041.387,7.429,-81.703,169.508,36.864,156.937
C01494=1041.381,7.179,-81.688,169.506,36.863,156.936
C01495=1041.374,6.930,-81.673,169.504,36.862,156.936
C01496=1041.367,6.681,-81.658,169.502,36.862,156.936
C01497=1041.362,6.431,-81.643,169.500,36.861,156.936
C01498=1041.356,6.182,-81.628,169.498,36.860,156.936
C01499=1041.349,5.933,-81.612,169.496,36.859,156.936
C01500=1041.343,5.683,-81.597,169.494,36.858,156.935
C01501=1041.337,5.433,-81.582,169.492,36.857,156.935
C01502=1041.330,5.184,-81.567,169.490,36.857,156.935
C01503=1041.324,4.935,-81.552,169.488,36.856,156.935
C01504=1041.317,4.685,-81.537,169.486,36.855,156.935
C01505=1041.311,4.435,-81.522,169.484,36.854,156.935
C01506=1041.305,4.186,-81.507,169.482,36.853,156.934
C01507=1041.299,3.937,-81.492,169.479,36.853,156.934
C01508=1041.292,3.688,-81.477,169.477,36.852,156.934
C01509=1041.286,3.438,-81.462,169.475,36.851,156.934
C01510=1041.280,3.188,-81.446,169.473,36.850,156.934
C01511=1041.273,2.938,-81.431,169.472,36.850,156.934
C01512=1041.267,2.689,-81.416,169.470,36.848,156.934
C01513=1041.261,2.440,-81.402,169.468,36.848,156.933
C01514=1041.255,2.191,-81.386,169.466,36.847,156.933
C01515=1041.248,1.941,-81.371,169.464,36.846,156.933
C01516=1041.242,1.691,-81.356,169.461,36.845,156.933
C01517=1041.235,1.442,-81.341,169.459,36.845,156.933
C01518=1041.230,1.193,-81.326,169.457,36.843,156.933
C01519=1041.223,0.943,-81.312,169.455,36.843,156.932
C01520=1041.217,0.693,-81.297,169.453,36.842,156.932
C01521=1041.211,0.444,-81.282,169.451,36.842,156.932
C01522=1041.204,0.194,-81.267,169.449,36.840,156.932
C01523=1041.198,-0.055,-81.252,169.447,36.840,156.932
C01524=1041.192,-0.305,-81.237,169.445,36.839,156.932
C01525=1041.185,-0.554,-81.222,169.443,36.838,156.931
C01526=1041.179,-0.803,-81.207,169.440,36.837,156.931
C01527=1041.173,-1.052,-81.192,169.438,36.837,156.931
C01528=1041.167,-1.302,-81.177,169.436,36.835,156.931
C01529=1041.160,-1.551,-81.162,169.435,36.835,156.931
C01530=1041.155,-1.801,-81.147,169.433,36.834,156.931
C01531=1041.149,-2.050,-81.132,169.431,36.833,156.931
C01532=1041.143,-2.300,-81.117,169.429,36.832,156.930
C01533=1041.136,-2.550,-81.102,169.427,36.832,156.930
C01534=1041.130,-2.799,-81.087,169.425,36.831,156.930
C01535=1041.123,-3.083,-81.071,169.423,36.830,156.930
C01536=1041.116,-3.366,-81.054,169.419,36.829,156.930
C01537=1041.109,-3.649,-81.037,169.417,36.828,156.930
C01538=1041.101,-3.933,-81.021,169.415,36.827,156.929
C01539=1041.095,-4.182,-81.006,169.413,36.827,156.929
C01540=1041.088,-4.432,-80.991,169.411,36.826,156.929
C01541=1041.082,-4.682,-80.976,169.409,36.825,156.929
C01542=1041.076,-4.931,-80.963,169.407,36.824,156.929
C01543=1041.069,-5.181,-80.948,169.405,36.823,156.929
C01544=1041.063,-5.430,-80.933,169.403,36.823,156.929
C01545=1041.057,-5.680,-80.918,169.401,36.822,156.928
C01546=1041.050,-5.929,-80.904,169.399,36.822,156.928
C01547=1041.044,-6.178,-80.889,169.396,36.821,156.928
C01548=1041.038,-6.428,-80.875,169.394,36.820,156.928
C01549=1041.031,-6.678,-80.861,169.392,36.820,156.928
C01550=1041.025,-6.927,-80.846,169.390,36.819,156.928
C01551=1041.018,-7.176,-80.831,169.388,36.818,156.928
C01552=1041.012,-7.426,-80.817,169.386,36.817,156.928
C01553=1041.006,-7.675,-80.803,169.384,36.817,156.927
C01554=1040.999,-7.925,-80.788,169.382,36.816,156.927
C01555=1040.993,-8.175,-80.773,169.380,36.815,156.927
C01556=1040.986,-8.424,-80.759,169.378,36.815,156.927
C01557=1040.980,-8.674,-80.745,169.376,36.814,156.927
C01558=1040.974,-8.923,-80.730,169.374,36.813,156.927
C01559=1040.967,-9.173,-80.715,169.371,36.813,156.927
C01560=1040.961,-9.422,-80.702,169.369,36.812,156.926
C01561=1040.955,-9.672,-80.687,169.367,36.811,156.926
C01562=1040.948,-9.921,-80.672,169.365,36.810,156.926
C01563=1040.942,-10.171,-80.658,169.363,36.810,156.926
C01564=1040.936,-10.420,-80.643,169.361,36.809,156.926
C01565=1040.930,-10.669,-80.629,169.359,36.808,156.926
C01566=1040.923,-10.919,-80.614,169.356,36.808,156.926
C01567=1040.917,-11.169,-80.600,169.354,36.807,156.926
C01568=1040.911,-11.418,-80.586,169.352,36.806,156.925
C01569=1040.905,-11.668,-80.572,169.350,36.805,156.925
C01570=1040.898,-11.918,-80.557,169.347,36.805,156.925
C01571=1040.892,-12.166,-80.543,169.345,36.804,156.925
C01572=1040.886,-12.416,-80.529,169.343,36.803,156.925
C01573=1040.880,-12.665,-80.514,169.341,36.803,156.925
C01574=1040.873,-12.915,-80.500,169.339,36.802,156.925
C01575=1040.867,-13.165,-80.486,169.337,36.801,156.925
C01576=1040.861,-13.414,-80.471,169.335,36.801,156.924
C01577=1040.854,-13.664,-80.458,169.333,36.800,156.924
C01578=1040.848,-13.913,-80.443,169.331,36.799,156.924
C01579=1040.842,-14.163,-80.429,169.329,36.798,156.924
C01580=1040.835,-14.413,-80.414,169.327,36.798,156.924
C01581=1040.829,-14.661,-80.400,169.325,36.797,156.924
C01582=1040.823,-14.912,-80.386,169.322,36.796,156.924
C01583=1040.817,-15.160,-80.372,169.320,36.796,156.923
C01584=1040.811,-15.411,-80.357,169.318,36.795,156.923
C01585=1040.804,-15.659,-80.343,169.316,36.795,156.923
C01586=1040.798,-15.910,-80.329,169.314,36.794,156.923
C01587=1040.791,-16.159,-80.315,169.312,36.793,156.923
C01588=1040.785,-16.409,-80.301,169.310,36.793,156.923
C01589=1040.779,-16.658,-80.287,169.308,36.792,156.923
C01590=1040.772,-16.907,-80.273,169.305,36.791,156.923
C01591=1040.766,-17.157,-80.259,169.303,36.791,156.922
C01592=1040.759,-17.406,-80.245,169.301,36.790,156.922
C01593=1040.753,-17.656,-80.231,169.299,36.790,156.922
C01594=1040.747,-17.906,-80.217,169.297,36.789,156.922
C01595=1040.740,-18.155,-80.203,169.294,36.788,156.922
C01596=1040.734,-18.405,-80.189,169.292,36.788,156.922
C01597=1040.727,-18.654,-80.175,169.290,36.787,156.922
C01598=1040.721,-18.904,-80.161,169.288,36.786,156.922
C01599=1040.714,-19.185,-80.145,169.285,36.786,156.922
C01600=1040.707,-19.468,-80.130,169.283,36.785,156.921
C01601=1040.700,-19.750,-80.114,169.281,36.785,156.921
C01602=1040.693,-20.031,-80.098,169.278,36.784,156.921
C01603=1040.686,-20.281,-80.084,169.276,36.783,156.921
C01604=1040.680,-20.530,-80.070,169.274,36.783,156.921
C01605=1040.674,-20.780,-80.057,169.272,36.782,156.921
C01606=1040.667,-21.029,-80.043,169.270,36.781,156.921
C01607=1040.661,-21.279,-80.028,169.268,36.781,156.921
C01608=1040.655,-21.528,-80.015,169.265,36.780,156.920
C01609=1040.648,-21.778,-80.000,169.263,36.780,156.920
C01610=1040.642,-22.027,-79.987,169.261,36.779,156.920
C01611=1040.635,-22.277,-79.973,169.259,36.778,156.920
C01612=1040.630,-22.527,-79.959,169.256,36.778,156.920
C01613=1040.623,-22.776,-79.945,169.254,36.777,156.920
C01614=1040.617,-23.025,-79.932,169.252,36.776,156.920
C01615=1040.611,-23.275,-79.918,169.250,36.776,156.920
C01616=1040.604,-23.525,-79.904,169.248,36.775,156.919
C01617=1040.599,-23.775,-79.890,169.246,36.775,156.919
C01618=1040.592,-24.024,-79.876,169.244,36.774,156.919
C01619=1040.585,-24.273,-79.863,169.242,36.773,156.919
C01620=1040.579,-24.523,-79.849,169.240,36.773,156.919
C01621=1040.573,-24.773,-79.835,169.238,36.773,156.919
C01622=1040.567,-25.022,-79.822,169.235,36.772,156.919
C01623=1040.561,-25.272,-79.807,169.232,36.771,156.919
C01624=1040.554,-25.521,-79.794,169.230,36.771,156.919
C01625=1040.548,-25.771,-79.780,169.228,36.770,156.919
C01626=1040.542,-26.020,-79.766,169.226,36.770,156.918
C01627=1040.536,-26.270,-79.753,169.224,36.769,156.918
C01628=1040.529,-26.520,-79.739,169.222,36.768,156.918
C01629=1040.524,-26.769,-79.726,169.220,36.768,156.918
C01630=1040.517,-27.018,-79.712,169.218,36.767,156.918
C01631=1040.510,-27.268,-79.698,169.215,36.766,156.918
C01632=1040.504,-27.517,-79.685,169.213,36.766,156.918
C01633=1040.497,-27.767,-79.671,169.211,36.766,156.918
C01634=1040.492,-28.017,-79.657,169.209,36.765,156.918
C01635=1040.486,-28.266,-79.644,169.207,36.765,156.917
C01636=1040.479,-28.516,-79.630,169.205,36.764,156.917
C01637=1040.473,-28.765,-79.617,169.201,36.763,156.917
C01638=1040.466,-29.015,-79.603,169.199,36.763,156.917
C01639=1040.459,-29.264,-79.590,169.197,36.763,156.917
C01640=1040.453,-29.514,-79.577,169.195,36.762,156.917
C01641=1040.446,-29.764,-79.563,169.193,36.761,156.917
C01642=1040.440,-30.013,-79.550,169.191,36.761,156.917
C01643=1040.435,-30.262,-79.536,169.189,36.761,156.917
C01644=1040.428,-30.512,-79.522,169.186,36.760,156.917
C01645=1040.422,-30.762,-79.509,169.184,36.760,156.916
C01646=1040.416,-31.011,-79.496,169.182,36.759,156.916
C01647=1040.409,-31.261,-79.483,169.180,36.758,156.916
C01648=1040.403,-31.511,-79.470,169.178,36.758,156.916
C01649=1040.397,-31.760,-79.456,169.176,36.758,156.916
C01650=1040.390,-32.010,-79.443,169.173,36.757,156.916
C01651=1040.384,-32.259,-79.430,169.171,36.756,156.916
C01652=1040.377,-32.508,-79.416,169.169,36.756,156.916
C01653=1040.371,-32.758,-79.403,169.167,36.756,156.916
C01654=1040.364,-33.008,-79.389,169.164,36.755,156.916
C01655=1040.358,-33.257,-79.376,169.162,36.754,156.916
C01656=1040.353,-33.507,-79.363,169.159,36.754,156.915
C01657=1040.346,-33.757,-79.349,169.157,36.754,156.915
C01658=1040.340,-34.006,-79.336,169.155,36.753,156.915
C01659=1040.334,-34.256,-79.323,169.153,36.753,156.915
C01660=1040.327,-34.505,-79.309,169.151,36.752,156.915
C01661=1040.321,-34.755,-79.296,169.148,36.751,156.915
C01662=1040.315,-35.005,-79.283,169.146,36.751,156.915
C01663=1040.307,-35.303,-79.267,169.144,36.751,156.915
C01664=1040.299,-35.602,-79.251,169.141,36.750,156.915
C01665=1040.292,-35.901,-79.235,169.138,36.749,156.915
C01666=1040.285,-36.200,-79.220,169.136,36.749,156.914
C01667=1040.278,-36.449,-79.206,169.134,36.748,156.914
C01668=1040.272,-36.698,-79.193,169.131,36.748,156.914
C01669=1040.266,-36.948,-79.180,169.129,36.748,156.914
C01670=1040.260,-37.198,-79.167,169.126,36.747,156.914
C01671=1040.254,-37.438,-79.154,169.124,36.746,156.914
C01672=1040.247,-37.679,-79.141,169.122,36.746,156.914
C01673=1040.242,-37.920,-79.129,169.120,36.746,156.914
C01674=1040.235,-38.161,-79.117,169.118,36.745,156.914
C01675=1040.230,-38.402,-79.104,169.116,36.744,156.914
C01676=1040.224,-38.642,-79.091,169.113,36.744,156.913
C01677=1040.218,-38.883,-79.078,169.111,36.744,156.913
C01678=1040.212,-39.124,-79.066,169.109,36.743,156.913
C01679=1040.205,-39.373,-79.054,169.107,36.743,156.913
C01680=1040.199,-39.622,-79.040,169.105,36.743,156.913
C01681=1040.192,-39.872,-79.027,169.102,36.742,156.913
C01682=1040.186,-40.122,-79.014,169.100,36.742,156.913
C01683=1040.180,-40.372,-79.001,169.098,36.741,156.913
C01684=1040.173,-40.621,-78.989,169.096,36.741,156.913
C01685=1040.167,-40.870,-78.976,169.093,36.741,156.913
C01686=1040.160,-41.120,-78.962,169.091,36.740,156.913
C01687=1040.155,-41.370,-78.949,169.089,36.740,156.913
C01688=1040.148,-41.619,-78.936,169.087,36.739,156.913
C01689=1040.142,-41.869,-78.924,169.085,36.739,156.913
C01690=1040.135,-42.118,-78.911,169.081,36.739,156.913
C01691=1040.130,-42.368,-78.898,169.079,36.738,156.912
C01692=1040.123,-42.617,-78.885,169.077,36.738,156.912
C01693=1040.117,-42.868,-78.872,169.075,36.738,156.912
C01694=1040.110,-43.117,-78.859,169.072,36.738,156.912
C01695=1040.104,-43.367,-78.847,169.070,36.737,156.912
C01696=1040.098,-43.616,-78.834,169.068,36.736,156.912
C01697=1040.092,-43.866,-78.821,169.066,36.736,156.912
C01698=1040.085,-44.115,-78.808,169.063,36.736,156.912
C01699=1040.079,-44.365,-78.796,169.061,36.736,156.912
C01700=1040.073,-44.614,-78.783,169.059,36.735,156.912
C01701=1040.067,-44.864,-78.770,169.057,36.734,156.912
C01702=1040.061,-45.114,-78.758,169.054,36.735,156.912
C01703=1040.053,-45.364,-78.744,169.052,36.734,156.912
C01704=1040.047,-45.613,-78.732,169.050,36.734,156.912
C01705=1040.041,-45.863,-78.719,169.048,36.733,156.911
C01706=1040.035,-46.113,-78.706,169.045,36.733,156.911
C01707=1040.028,-46.362,-78.693,169.043,36.733,156.911
C01708=1040.022,-46.611,-78.681,169.041,36.732,156.911
C01709=1040.017,-46.861,-78.668,169.039,36.732,156.911
C01710=1040.010,-47.111,-78.655,169.036,36.731,156.911
C01711=1040.004,-47.360,-78.643,169.034,36.731,156.911
C01712=1039.998,-47.610,-78.631,169.031,36.731,156.911
C01713=1039.992,-47.859,-78.617,169.029,36.730,156.911
C01714=1039.985,-48.109,-78.605,169.026,36.730,156.911
C01715=1039.979,-48.359,-78.593,169.024,36.730,156.911
C01716=1039.973,-48.608,-78.579,169.022,36.730,156.911
C01717=1039.967,-48.858,-78.567,169.019,36.729,156.911
C01718=1039.960,-49.107,-78.555,169.017,36.729,156.911
C01719=1039.954,-49.357,-78.542,169.015,36.728,156.910
C01720=1039.948,-49.607,-78.529,169.013,36.728,156.910
C01721=1039.942,-49.856,-78.517,169.010,36.728,156.910
C01722=1039.936,-50.106,-78.505,169.008,36.727,156.910
C01723=1039.929,-50.355,-78.491,169.006,36.727,156.910
C01724=1039.923,-50.605,-78.479,169.004,36.726,156.910
C01725=1039.917,-50.855,-78.467,169.001,36.726,156.910
C01726=1039.910,-51.104,-78.455,168.999,36.726,156.910
C01727=1039.903,-51.386,-78.440,168.996,36.726,156.910
C01728=1039.896,-51.668,-78.427,168.994,36.726,156.910
C01729=1039.889,-51.949,-78.413,168.991,36.726,156.910
C01730=1039.882,-52.231,-78.399,168.988,36.725,156.910
C01731=1039.875,-52.480,-78.387,168.986,36.725,156.910
C01732=1039.868,-52.729,-78.374,168.984,36.725,156.910
C01733=1039.862,-52.979,-78.362,168.981,36.725,156.910
C01734=1039.856,-53.229,-78.350,168.979,36.725,156.910
C01735=1039.850,-53.478,-78.337,168.977,36.725,156.910
C01736=1039.843,-53.728,-78.325,168.974,36.724,156.910
C01737=1039.837,-53.978,-78.313,168.972,36.724,156.910
C01738=1039.831,-54.227,-78.301,168.970,36.724,156.910
C01739=1039.824,-54.477,-78.289,168.967,36.723,156.909
C01740=1039.817,-54.727,-78.277,168.965,36.723,156.909
C01741=1039.812,-54.976,-78.264,168.963,36.723,156.909
C01742=1039.805,-55.226,-78.252,168.960,36.723,156.909
C01743=1039.798,-55.476,-78.240,168.957,36.723,156.909
C01744=1039.792,-55.726,-78.228,168.955,36.723,156.909
C01745=1039.786,-55.975,-78.216,168.952,36.723,156.909
C01746=1039.780,-56.224,-78.204,168.950,36.722,156.909
C01747=1039.774,-56.474,-78.192,168.948,36.722,156.909
C01748=1039.767,-56.723,-78.180,168.945,36.722,156.909
C01749=1039.761,-56.973,-78.167,168.943,36.722,156.909
C01750=1039.755,-57.223,-78.155,168.941,36.722,156.909
C01751=1039.748,-57.472,-78.143,168.938,36.722,156.909
C01752=1039.742,-57.722,-78.131,168.936,36.722,156.909
C01753=1039.735,-57.972,-78.119,168.934,36.721,156.909
C01754=1039.729,-58.221,-78.107,168.931,36.721,156.909
C01755=1039.723,-58.471,-78.095,168.929,36.721,156.909
C01756=1039.717,-58.720,-78.083,168.926,36.721,156.909
C01757=1039.710,-58.970,-78.071,168.924,36.720,156.909
C01758=1039.704,-59.220,-78.058,168.922,36.720,156.909
C01759=1039.698,-59.469,-78.046,168.919,36.720,156.909
C01760=1039.691,-59.719,-78.034,168.917,36.720,156.909
C01761=1039.685,-59.969,-78.022,168.915,36.720,156.909
C01762=1039.679,-60.218,-78.011,168.912,36.720,156.909
C01763=1039.673,-60.468,-77.999,168.910,36.720,156.909
C01764=1039.666,-60.717,-77.987,168.908,36.719,156.909
C01765=1039.660,-60.967,-77.974,168.905,36.719,156.909
C01766=1039.653,-61.217,-77.962,168.903,36.719,156.909
C01767=1039.648,-61.466,-77.952,168.901,36.719,156.909
C01768=1039.642,-61.716,-77.939,168.898,36.719,156.908
C01769=1039.635,-61.966,-77.927,168.896,36.719,156.908
C01770=1039.628,-62.215,-77.915,168.893,36.719,156.908
C01771=1039.623,-62.465,-77.902,168.891,36.719,156.908
C01772=1039.616,-62.714,-77.891,168.889,36.718,156.908
C01773=1039.610,-62.964,-77.880,168.886,36.718,156.908
C01774=1039.604,-63.214,-77.867,168.884,36.718,156.908
C01775=1039.598,-63.464,-77.855,168.882,36.718,156.908
C01776=1039.592,-63.713,-77.844,168.879,36.717,156.908
C01777=1039.585,-63.963,-77.832,168.877,36.717,156.908
C01778=1039.579,-64.213,-77.820,168.874,36.717,156.908
C01779=1039.573,-64.462,-77.808,168.872,36.717,156.908
C01780=1039.567,-64.711,-77.796,168.870,36.717,156.908
C01781=1039.561,-64.962,-77.784,168.867,36.717,156.908
C01782=1039.554,-65.211,-77.772,168.865,36.717,156.908
C01783=1039.548,-65.460,-77.761,168.863,36.717,156.908
C01784=1039.542,-65.710,-77.750,168.860,36.717,156.908
C01785=1039.536,-65.960,-77.737,168.858,36.716,156.908
C01786=1039.529,-66.210,-77.725,168.855,36.716,156.908
C01787=1039.524,-66.459,-77.714,168.853,36.716,156.908
C01788=1039.517,-66.709,-77.702,168.851,36.716,156.908
C01789=1039.511,-66.959,-77.690,168.848,36.716,156.908
C01790=1039.505,-67.208,-77.679,168.846,36.716,156.908
C01791=1039.498,-67.491,-77.665,168.843,36.716,156.908
C01792=1039.491,-67.774,-77.652,168.841,36.716,156.908
C01793=1039.484,-68.056,-77.639,168.837,36.715,156.908
C01794=1039.477,-68.339,-77.626,168.834,36.715,156.908
C01795=1039.471,-68.588,-77.614,168.832,36.715,156.908
C01796=1039.465,-68.839,-77.602,168.829,36.715,156.908
C01797=1039.459,-69.088,-77.590,168.827,36.715,156.908
C01798=1039.453,-69.338,-77.579,168.825,36.714,156.908
C01799=1039.446,-69.588,-77.567,168.822,36.714,156.908
C01800=1039.441,-69.837,-77.556,168.820,36.714,156.908
C01801=1039.435,-70.087,-77.544,168.817,36.714,156.908
C01802=1039.429,-70.336,-77.532,168.815,36.714,156.908
C01803=1039.422,-70.586,-77.521,168.813,36.714,156.908
C01804=1039.416,-70.836,-77.509,168.810,36.714,156.907
C01805=1039.411,-71.085,-77.497,168.808,36.714,156.907
C01806=1039.404,-71.335,-77.485,168.805,36.714,156.907
